LIN {X 0,Y 292.051,Z 857.28,A -85,B 0,C 180,E1 15092.157,E2 15092.157} C_VEL
LIN {X 0,Y 292.417,Z 857.28,A -85,B 0,C 180,E1 15098.753,E2 15098.753} C_VEL
LIN {X 0,Y 292.75,Z 857.28,A -85,B 0,C 180,E1 15104.981,E2 15104.981} C_VEL
LIN {X 0,Y 293.457,Z 857.28,A -85,B 0,C 180,E1 15114.042,E2 15114.042} C_VEL
LIN {X 0,Y 293.996,Z 857.28,A -85,B 0,C 180,E1 15119.962,E2 15119.962} C_VEL
LIN {X 0,Y 293.479,Z 857.28,A -85,B 0,C 180,E1 15125.882,E2 15125.882} C_VEL
LIN {X 0,Y 293.039,Z 857.28,A -85,B 0,C 180,E1 15131.883,E2 15131.883} C_VEL
LIN {X 0,Y 292.64,Z 857.28,A -85,B 0,C 180,E1 15138.037,E2 15138.037} C_VEL
LIN {X 0,Y 292.24,Z 857.28,A -85,B 0,C 180,E1 15144.433,E2 15144.433} C_VEL
LIN {X 0,Y 291.833,Z 857.307,A -85,B 0,C 180,E1 15152.49,E2 15152.49} C_VEL
LIN {X 0,Y 294.082,Z 862.737,A -85,B 0,C 180,E1 15153.268,E2 15153.268} C_VEL
LIN {X 0,Y 306.27,Z 885.121,A -85,B 0,C 180,E1 15157.392,E2 15157.392} C_VEL
LIN {X 0,Y 314.782,Z 908.516,A -85,B 0,C 180,E1 15161.429,E2 15161.429} C_VEL
LIN {X 0,Y 318.92,Z 932.003,A -85,B 0,C 180,E1 15165.576,E2 15165.576} C_VEL
LIN {X 0,Y 315.348,Z 948.213,A -85,B 0,C 180,E1 15168.226,E2 15168.226} C_VEL
LIN {X 0,Y 308.77,Z 968.688,A -85,B 0,C 180,E1 15172.765,E2 15172.765} C_VEL
LIN {X 0,Y 303.225,Z 983.739,A -85,B 0,C 180,E1 15177.978,E2 15177.978} C_VEL
LIN {X 0,Y 299.821,Z 992.395,A -85,B 0,C 180,E1 15182.966,E2 15182.966} C_VEL
LIN {X 0,Y 297.402,Z 997.125,A -85,B 0,C 180,E1 15189.121,E2 15189.121} C_VEL
LIN {X 0,Y 296.865,Z 995.934,A -85,B 0,C 180,E1 15195.459,E2 15195.459} C_VEL
LIN {X 0,Y 298.171,Z 989.36,A -85,B 0,C 180,E1 15201.237,E2 15201.237} C_VEL
LIN {X 0,Y 300.527,Z 978.42,A -85,B 0,C 180,E1 15206.388,E2 15206.388} C_VEL
LIN {X 0,Y 304.232,Z 961.601,A -85,B 0,C 180,E1 15211.425,E2 15211.425} C_VEL
LIN {X 0,Y 308.992,Z 939.449,A -85,B 0,C 180,E1 15215.799,E2 15215.799} C_VEL
LIN {X 0,Y 311.298,Z 922.827,A -85,B 0,C 180,E1 15218.213,E2 15218.213} C_VEL
LIN {X 0,Y 307.426,Z 899.704,A -85,B 0,C 180,E1 15221.361,E2 15221.361} C_VEL
LIN {X 0,Y 298.936,Z 872.735,A -85,B 0,C 180,E1 15224.452,E2 15224.452} C_VEL
LIN {X 0,Y 292.791,Z 857.28,A -85,B 0,C 180,E1 15226.014,E2 15226.014} C_VEL
LIN {X 0,Y 292.167,Z 857.28,A -85,B 0,C 180,E1 15234.492,E2 15234.492} C_VEL
LIN {X 0,Y 291.84,Z 857.28,A -85,B 0,C 180,E1 15241.251,E2 15241.251} C_VEL
LIN {X 0,Y 291.876,Z 857.28,A -85,B 0,C 180,E1 15249.731,E2 15249.731} C_VEL
LIN {X 0,Y 301.053,Z 889.147,A -85,B 0,C 180,E1 15251.908,E2 15251.908} C_VEL
LIN {X 0,Y 306.355,Z 915.006,A -85,B 0,C 180,E1 15254.516,E2 15254.516} C_VEL
LIN {X 0,Y 304.215,Z 939.148,A -85,B 0,C 180,E1 15257.526,E2 15257.526} C_VEL
LIN {X 0,Y 301.338,Z 961.008,A -85,B 0,C 180,E1 15261.49,E2 15261.49} C_VEL
LIN {X 0,Y 298.964,Z 978.431,A -85,B 0,C 180,E1 15266.207,E2 15266.207} C_VEL
LIN {X 0,Y 297.475,Z 990.318,A -85,B 0,C 180,E1 15271.29,E2 15271.29} C_VEL
LIN {X 0,Y 296.907,Z 996.961,A -85,B 0,C 180,E1 15276.62,E2 15276.62} C_VEL
LIN {X 0,Y 297.738,Z 998.146,A -85,B 0,C 180,E1 15282.282,E2 15282.282} C_VEL
LIN {X 0,Y 299.876,Z 993.695,A -85,B 0,C 180,E1 15287.652,E2 15287.652} C_VEL
LIN {X 0,Y 303.37,Z 983.119,A -85,B 0,C 180,E1 15293.016,E2 15293.016} C_VEL
LIN {X 0,Y 307.54,Z 967.861,A -85,B 0,C 180,E1 15297.568,E2 15297.568} C_VEL
LIN {X 0,Y 312.162,Z 947.905,A -85,B 0,C 180,E1 15301.439,E2 15301.439} C_VEL
LIN {X 0,Y 316.12,Z 922.658,A -85,B 0,C 180,E1 15304.704,E2 15304.704} C_VEL
LIN {X 0,Y 312.93,Z 899.843,A -85,B 0,C 180,E1 15307.526,E2 15307.526} C_VEL
LIN {X 0,Y 304.863,Z 879.144,A -85,B 0,C 180,E1 15310.308,E2 15310.308} C_VEL
LIN {X 0,Y 295.138,Z 862.737,A -85,B 0,C 180,E1 15313.251,E2 15313.251} C_VEL
LIN {X 0,Y 292.877,Z 857.28,A -85,B 0,C 180,E1 15314.248,E2 15314.248} C_VEL
LIN {X 0,Y 292.427,Z 857.28,A -85,B 0,C 180,E1 15321.281,E2 15321.281} C_VEL
LIN {X 0,Y 292.014,Z 857.28,A -85,B 0,C 180,E1 15328.186,E2 15328.186} C_VEL
LIN {X 0,Y 291.802,Z 857.28,A -85,B 0,C 180,E1 15334.832,E2 15334.832} C_VEL
LIN {X 0,Y 291.583,Z 857.28,A -85,B 0,C 180,E1 15343.369,E2 15343.369} C_VEL
LIN {X 0,Y 291.824,Z 857.28,A -85,B 0,C 180,E1 15347.489,E2 15347.489} C_VEL
LIN {X 0,Y 313.414,Z 909.451,A -85,B 0,C 180,E1 15351.464,E2 15351.464} C_VEL
LIN {X 0,Y 320.249,Z 933.058,A -85,B 0,C 180,E1 15353.265,E2 15353.265} C_VEL
LIN {X 0,Y 315.373,Z 966.492,A -85,B 0,C 180,E1 15355.452,E2 15355.452} C_VEL
LIN {X 0,Y 309.547,Z 998.009,A -85,B 0,C 180,E1 15358.778,E2 15358.778} C_VEL
LIN {X 0,Y 303.847,Z 1024.876,A -85,B 0,C 180,E1 15362.955,E2 15362.955} C_VEL
LIN {X 0,Y 299.229,Z 1047.786,A -85,B 0,C 180,E1 15368.09,E2 15368.09} C_VEL
LIN {X 0,Y 296.572,Z 1065.205,A -85,B 0,C 180,E1 15373.694,E2 15373.694} C_VEL
LIN {X 0,Y 295.641,Z 1077.565,A -85,B 0,C 180,E1 15379.675,E2 15379.675} C_VEL
LIN {X 0,Y 295.789,Z 1083.188,A -85,B 0,C 180,E1 15384.125,E2 15384.125} C_VEL
LIN {X 0,Y 296.066,Z 1086.174,A -85,B 0,C 180,E1 15390.001,E2 15390.001} C_VEL
LIN {X 0,Y 295.708,Z 1084.155,A -85,B 0,C 180,E1 15395.879,E2 15395.879} C_VEL
LIN {X 0,Y 295.5,Z 1077.25,A -85,B 0,C 180,E1 15401.828,E2 15401.828} C_VEL
LIN {X 0,Y 297.243,Z 1063.717,A -85,B 0,C 180,E1 15408.399,E2 15408.399} C_VEL
LIN {X 0,Y 301.566,Z 1044.337,A -85,B 0,C 180,E1 15414.543,E2 15414.543} C_VEL
LIN {X 0,Y 307.998,Z 1020.257,A -85,B 0,C 180,E1 15419.758,E2 15419.758} C_VEL
LIN {X 0,Y 315.4,Z 992.25,A -85,B 0,C 180,E1 15423.923,E2 15423.923} C_VEL
LIN {X 0,Y 322.553,Z 960.566,A -85,B 0,C 180,E1 15427.038,E2 15427.038} C_VEL
LIN {X 0,Y 326.962,Z 932.174,A -85,B 0,C 180,E1 15428.868,E2 15428.868} C_VEL
LIN {X 0,Y 318.461,Z 906.2,A -85,B 0,C 180,E1 15431.59,E2 15431.59} C_VEL
LIN {X 0,Y 317.145,Z 903.31,A -85,B 0,C 180,E1 15431.93,E2 15431.93} C_VEL
LIN {X 0,Y 310.668,Z 894.982,A -85,B 0,C 180,E1 15433.356,E2 15433.356} C_VEL
LIN {X 0,Y 299.831,Z 884.402,A -85,B 0,C 180,E1 15435.807,E2 15435.807} C_VEL
LIN {X 0,Y 298.921,Z 882.832,A -85,B 0,C 180,E1 15436.05,E2 15436.05} C_VEL
LIN {X 0,Y 286.284,Z 862.993,A -85,B 0,C 180,E1 15439.689,E2 15439.689} C_VEL
LIN {X 0,Y 283.795,Z 857.28,A -85,B 0,C 180,E1 15440.762,E2 15440.762} C_VEL
LIN {X 0,Y 283.97,Z 857.28,A -85,B 0,C 180,E1 15448.552,E2 15448.552} C_VEL
LIN {X 0,Y 284.238,Z 857.28,A -85,B 0,C 180,E1 15454.901,E2 15454.901} C_VEL
LIN {X 0,Y 284.673,Z 857.28,A -85,B 0,C 180,E1 15463.211,E2 15463.211} C_VEL
LIN {X 0,Y 285.234,Z 857.28,A -85,B 0,C 180,E1 15470.801,E2 15470.801} C_VEL
LIN {X 0,Y 285.877,Z 857.28,A -85,B 0,C 180,E1 15476.927,E2 15476.927} C_VEL
LIN {X 0,Y 285.868,Z 857.28,A -85,B 0,C 180,E1 15482.996,E2 15482.996} C_VEL
LIN {X 0,Y 285.075,Z 857.28,A -85,B 0,C 180,E1 15492.22,E2 15492.22} C_VEL
LIN {X 0,Y 284.66,Z 857.28,A -85,B 0,C 180,E1 15498.561,E2 15498.561} C_VEL
LIN {X 0,Y 284.213,Z 857.28,A -85,B 0,C 180,E1 15505.171,E2 15505.171} C_VEL
LIN {X 0,Y 283.965,Z 857.28,A -85,B 0,C 180,E1 15510.494,E2 15510.494} C_VEL
LIN {X 0,Y 286.238,Z 862.79,A -85,B 0,C 180,E1 15511.368,E2 15511.368} C_VEL
LIN {X 0,Y 298.239,Z 884.055,A -85,B 0,C 180,E1 15515.658,E2 15515.658} C_VEL
LIN {X 0,Y 307.422,Z 908.201,A -85,B 0,C 180,E1 15520.086,E2 15520.086} C_VEL
LIN {X 0,Y 311.823,Z 930.492,A -85,B 0,C 180,E1 15524.182,E2 15524.182} C_VEL
LIN {X 0,Y 311.465,Z 939.871,A -85,B 0,C 180,E1 15525.876,E2 15525.876} C_VEL
LIN {X 0,Y 304.54,Z 962.032,A -85,B 0,C 180,E1 15530.089,E2 15530.089} C_VEL
LIN {X 0,Y 298.43,Z 978.637,A -85,B 0,C 180,E1 15534.895,E2 15534.895} C_VEL
LIN {X 0,Y 293.676,Z 990.339,A -85,B 0,C 180,E1 15540.308,E2 15540.308} C_VEL
LIN {X 0,Y 290.878,Z 996.46,A -85,B 0,C 180,E1 15545.39,E2 15545.39} C_VEL
LIN {X 0,Y 289.12,Z 998.561,A -85,B 0,C 180,E1 15551.686,E2 15551.686} C_VEL
LIN {X 0,Y 289.394,Z 995.02,A -85,B 0,C 180,E1 15557.919,E2 15557.919} C_VEL
LIN {X 0,Y 291.487,Z 985.654,A -85,B 0,C 180,E1 15564.036,E2 15564.036} C_VEL
LIN {X 0,Y 294.927,Z 970.748,A -85,B 0,C 180,E1 15569.638,E2 15569.638} C_VEL
LIN {X 0,Y 299.377,Z 951.389,A -85,B 0,C 180,E1 15574.35,E2 15574.35} C_VEL
LIN {X 0,Y 304.25,Z 927.681,A -85,B 0,C 180,E1 15578.225,E2 15578.225} C_VEL
LIN {X 0,Y 300.861,Z 904.233,A -85,B 0,C 180,E1 15581.612,E2 15581.612} C_VEL
LIN {X 0,Y 292.909,Z 877.335,A -85,B 0,C 180,E1 15584.884,E2 15584.884} C_VEL
LIN {X 0,Y 284.754,Z 857.28,A -85,B 0,C 180,E1 15587.062,E2 15587.062} C_VEL
LIN {X 0,Y 284.152,Z 857.28,A -85,B 0,C 180,E1 15595.23,E2 15595.23} C_VEL
LIN {X 0,Y 283.876,Z 857.28,A -85,B 0,C 180,E1 15602.231,E2 15602.231} C_VEL
LIN {X 0,Y 283.938,Z 857.591,A -85,B 0,C 180,E1 15609.114,E2 15609.114} C_VEL
LIN {X 0,Y 292.917,Z 887.919,A -85,B 0,C 180,E1 15611.226,E2 15611.226} C_VEL
LIN {X 0,Y 298.57,Z 914.947,A -85,B 0,C 180,E1 15613.964,E2 15613.964} C_VEL
LIN {X 0,Y 297.666,Z 932.003,A -85,B 0,C 180,E1 15616.014,E2 15616.014} C_VEL
LIN {X 0,Y 294.567,Z 955.511,A -85,B 0,C 180,E1 15619.844,E2 15619.844} C_VEL
LIN {X 0,Y 291.757,Z 975.193,A -85,B 0,C 180,E1 15624.652,E2 15624.652} C_VEL
LIN {X 0,Y 290.044,Z 988.276,A -85,B 0,C 180,E1 15629.582,E2 15629.582} C_VEL
LIN {X 0,Y 289.1,Z 996.941,A -85,B 0,C 180,E1 15635.284,E2 15635.284} C_VEL
LIN {X 0,Y 289.475,Z 999.663,A -85,B 0,C 180,E1 15640.298,E2 15640.298} C_VEL
LIN {X 0,Y 291.556,Z 996.856,A -85,B 0,C 180,E1 15646.531,E2 15646.531} C_VEL
LIN {X 0,Y 294.757,Z 988.441,A -85,B 0,C 180,E1 15651.921,E2 15651.921} C_VEL
LIN {X 0,Y 299.092,Z 974.706,A -85,B 0,C 180,E1 15656.813,E2 15656.813} C_VEL
LIN {X 0,Y 304.047,Z 955.73,A -85,B 0,C 180,E1 15661.098,E2 15661.098} C_VEL
LIN {X 0,Y 308.919,Z 931.93,A -85,B 0,C 180,E1 15664.602,E2 15664.602} C_VEL
LIN {X 0,Y 309.271,Z 917.044,A -85,B 0,C 180,E1 15666.479,E2 15666.479} C_VEL
LIN {X 0,Y 304.585,Z 894.987,A -85,B 0,C 180,E1 15669.387,E2 15669.387} C_VEL
LIN {X 0,Y 294.414,Z 874.073,A -85,B 0,C 180,E1 15672.781,E2 15672.781} C_VEL
LIN {X 0,Y 287.331,Z 863.007,A -85,B 0,C 180,E1 15675.309,E2 15675.309} C_VEL
LIN {X 0,Y 284.773,Z 857.873,A -85,B 0,C 180,E1 15676.446,E2 15676.446} C_VEL
LIN {X 0,Y 284.247,Z 857.28,A -85,B 0,C 180,E1 15685.254,E2 15685.254} C_VEL
LIN {X 0,Y 283.918,Z 857.28,A -85,B 0,C 180,E1 15692.258,E2 15692.258} C_VEL
LIN {X 0,Y 283.636,Z 857.28,A -85,B 0,C 180,E1 15699.865,E2 15699.865} C_VEL
LIN {X 0,Y 283.896,Z 857.417,A -85,B 0,C 180,E1 15706.478,E2 15706.478} C_VEL
LIN {X 0,Y 305.889,Z 909.715,A -85,B 0,C 180,E1 15710.687,E2 15710.687} C_VEL
LIN {X 0,Y 313.023,Z 934.811,A -85,B 0,C 180,E1 15712.692,E2 15712.692} C_VEL
LIN {X 0,Y 308.007,Z 967.343,A -85,B 0,C 180,E1 15714.935,E2 15714.935} C_VEL
LIN {X 0,Y 302.051,Z 998.129,A -85,B 0,C 180,E1 15718.313,E2 15718.313} C_VEL
LIN {X 0,Y 296.162,Z 1024.75,A -85,B 0,C 180,E1 15722.607,E2 15722.607} C_VEL
LIN {X 0,Y 291.415,Z 1047.459,A -85,B 0,C 180,E1 15727.873,E2 15727.873} C_VEL
LIN {X 0,Y 288.578,Z 1065.563,A -85,B 0,C 180,E1 15734.012,E2 15734.012} C_VEL
LIN {X 0,Y 287.802,Z 1077.356,A -85,B 0,C 180,E1 15740.156,E2 15740.156} C_VEL
LIN {X 0,Y 287.912,Z 1083.164,A -85,B 0,C 180,E1 15745.477,E2 15745.477} C_VEL
LIN {X 0,Y 288.249,Z 1084.978,A -85,B 0,C 180,E1 15750.001,E2 15750.001} C_VEL
LIN {X 0,Y 287.855,Z 1083.014,A -85,B 0,C 180,E1 15756.04,E2 15756.04} C_VEL
LIN {X 0,Y 287.661,Z 1076.153,A -85,B 0,C 180,E1 15762.155,E2 15762.155} C_VEL
LIN {X 0,Y 289.488,Z 1063.13,A -85,B 0,C 180,E1 15768.729,E2 15768.729} C_VEL
LIN {X 0,Y 293.872,Z 1044.632,A -85,B 0,C 180,E1 15774.869,E2 15774.869} C_VEL
LIN {X 0,Y 300.588,Z 1020.977,A -85,B 0,C 180,E1 15780.247,E2 15780.247} C_VEL
LIN {X 0,Y 308.41,Z 992.884,A -85,B 0,C 180,E1 15784.587,E2 15784.587} C_VEL
LIN {X 0,Y 315.859,Z 961.774,A -85,B 0,C 180,E1 15787.763,E2 15787.763} C_VEL
LIN {X 0,Y 320.588,Z 934.743,A -85,B 0,C 180,E1 15789.585,E2 15789.585} C_VEL
LIN {X 0,Y 312.809,Z 909.957,A -85,B 0,C 180,E1 15792.355,E2 15792.355} C_VEL
LIN {X 0,Y 298.921,Z 882.832,A -85,B 0,C 180,E1 15796.05,E2 15796.05} C_VEL
LIN {X 0,Y 294.151,Z 878.708,A -85,B 0,C 180,E1 15797.228,E2 15797.228} C_VEL
LIN {X 0,Y 286.224,Z 874.597,A -85,B 0,C 180,E1 15799.245,E2 15799.245} C_VEL
LIN {X 0,Y 285.555,Z 873.708,A -85,B 0,C 180,E1 15799.446,E2 15799.446} C_VEL
LIN {X 0,Y 278.339,Z 862.989,A -85,B 0,C 180,E1 15801.827,E2 15801.827} C_VEL
LIN {X 0,Y 275.912,Z 858.523,A -85,B 0,C 180,E1 15802.729,E2 15802.729} C_VEL
LIN {X 0,Y 275.812,Z 857.28,A -85,B 0,C 180,E1 15802.822,E2 15802.822} C_VEL
LIN {X 0,Y 276.138,Z 857.28,A -85,B 0,C 180,E1 15811.319,E2 15811.319} C_VEL
LIN {X 0,Y 276.489,Z 857.28,A -85,B 0,C 180,E1 15818.584,E2 15818.584} C_VEL
LIN {X 0,Y 276.987,Z 857.28,A -85,B 0,C 180,E1 15827.335,E2 15827.335} C_VEL
LIN {X 0,Y 277.571,Z 857.28,A -85,B 0,C 180,E1 15833.699,E2 15833.699} C_VEL
LIN {X 0,Y 278.214,Z 857.28,A -85,B 0,C 180,E1 15839.96,E2 15839.96} C_VEL
LIN {X 0,Y 277.596,Z 857.28,A -85,B 0,C 180,E1 15846.22,E2 15846.22} C_VEL
LIN {X 0,Y 277.106,Z 857.28,A -85,B 0,C 180,E1 15852.578,E2 15852.578} C_VEL
LIN {X 0,Y 276.528,Z 857.28,A -85,B 0,C 180,E1 15861.436,E2 15861.436} C_VEL
LIN {X 0,Y 276.144,Z 857.447,A -85,B 0,C 180,E1 15868.317,E2 15868.317} C_VEL
LIN {X 0,Y 278.394,Z 862.813,A -85,B 0,C 180,E1 15869.246,E2 15869.246} C_VEL
LIN {X 0,Y 287.831,Z 878.44,A -85,B 0,C 180,E1 15872.812,E2 15872.812} C_VEL
LIN {X 0,Y 297.594,Z 899.927,A -85,B 0,C 180,E1 15877.132,E2 15877.132} C_VEL
LIN {X 0,Y 303.904,Z 923.425,A -85,B 0,C 180,E1 15881.64,E2 15881.64} C_VEL
LIN {X 0,Y 305.296,Z 940.028,A -85,B 0,C 180,E1 15884.9,E2 15884.9} C_VEL
LIN {X 0,Y 298.158,Z 962.047,A -85,B 0,C 180,E1 15889.086,E2 15889.086} C_VEL
LIN {X 0,Y 291.512,Z 979.299,A -85,B 0,C 180,E1 15894.083,E2 15894.083} C_VEL
LIN {X 0,Y 286.545,Z 990.786,A -85,B 0,C 180,E1 15899.357,E2 15899.357} C_VEL
LIN {X 0,Y 283.159,Z 997.767,A -85,B 0,C 180,E1 15905.22,E2 15905.22} C_VEL
LIN {X 0,Y 281.371,Z 999.797,A -85,B 0,C 180,E1 15911.163,E2 15911.163} C_VEL
LIN {X 0,Y 281.504,Z 996.586,A -85,B 0,C 180,E1 15917.575,E2 15917.575} C_VEL
LIN {X 0,Y 283.583,Z 987.566,A -85,B 0,C 180,E1 15923.869,E2 15923.869} C_VEL
LIN {X 0,Y 287.003,Z 973.119,A -85,B 0,C 180,E1 15929.621,E2 15929.621} C_VEL
LIN {X 0,Y 291.516,Z 954.311,A -85,B 0,C 180,E1 15934.467,E2 15934.467} C_VEL
LIN {X 0,Y 296.78,Z 930.157,A -85,B 0,C 180,E1 15938.618,E2 15938.618} C_VEL
LIN {X 0,Y 294.256,Z 908.622,A -85,B 0,C 180,E1 15941.876,E2 15941.876} C_VEL
LIN {X 0,Y 286.962,Z 882.251,A -85,B 0,C 180,E1 15945.295,E2 15945.295} C_VEL
LIN {X 0,Y 276.717,Z 857.28,A -85,B 0,C 180,E1 15948.168,E2 15948.168} C_VEL
LIN {X 0,Y 276.119,Z 857.28,A -85,B 0,C 180,E1 15956.018,E2 15956.018} C_VEL
LIN {X 0,Y 275.743,Z 857.28,A -85,B 0,C 180,E1 15964.657,E2 15964.657} C_VEL
LIN {X 0,Y 275.968,Z 857.28,A -85,B 0,C 180,E1 15968.419,E2 15968.419} C_VEL
LIN {X 0,Y 285.494,Z 889.664,A -85,B 0,C 180,E1 15970.765,E2 15970.765} C_VEL
LIN {X 0,Y 291.2,Z 917.429,A -85,B 0,C 180,E1 15973.701,E2 15973.701} C_VEL
LIN {X 0,Y 288.925,Z 941.854,A -85,B 0,C 180,E1 15976.917,E2 15976.917} C_VEL
LIN {X 0,Y 285.705,Z 964.372,A -85,B 0,C 180,E1 15981.246,E2 15981.246} C_VEL
LIN {X 0,Y 283.381,Z 980.958,A -85,B 0,C 180,E1 15986.028,E2 15986.028} C_VEL
LIN {X 0,Y 281.845,Z 992.463,A -85,B 0,C 180,E1 15991.146,E2 15991.146} C_VEL
LIN {X 0,Y 281.271,Z 998.914,A -85,B 0,C 180,E1 15996.218,E2 15996.218} C_VEL
LIN {X 0,Y 281.876,Z 1001.013,A -85,B 0,C 180,E1 16001.249,E2 16001.249} C_VEL
LIN {X 0,Y 283.6,Z 998.938,A -85,B 0,C 180,E1 16006.145,E2 16006.145} C_VEL
LIN {X 0,Y 286.889,Z 991.422,A -85,B 0,C 180,E1 16011.698,E2 16011.698} C_VEL
LIN {X 0,Y 291.641,Z 977.605,A -85,B 0,C 180,E1 16017.063,E2 16017.063} C_VEL
LIN {X 0,Y 297.012,Z 958.793,A -85,B 0,C 180,E1 16021.567,E2 16021.567} C_VEL
LIN {X 0,Y 302.322,Z 935.135,A -85,B 0,C 180,E1 16025.243,E2 16025.243} C_VEL
LIN {X 0,Y 303.209,Z 921.956,A -85,B 0,C 180,E1 16026.947,E2 16026.947} C_VEL
LIN {X 0,Y 299.526,Z 900.362,A -85,B 0,C 180,E1 16029.954,E2 16029.954} C_VEL
LIN {X 0,Y 290.435,Z 880.101,A -85,B 0,C 180,E1 16033.405,E2 16033.405} C_VEL
LIN {X 0,Y 283.088,Z 868.605,A -85,B 0,C 180,E1 16036.212,E2 16036.212} C_VEL
LIN {X 0,Y 279.789,Z 863.502,A -85,B 0,C 180,E1 16037.708,E2 16037.708} C_VEL
LIN {X 0,Y 276.691,Z 858.449,A -85,B 0,C 180,E1 16039.338,E2 16039.338} C_VEL
LIN {X 0,Y 276.551,Z 857.28,A -85,B 0,C 180,E1 16039.762,E2 16039.762} C_VEL
LIN {X 0,Y 276.14,Z 857.28,A -85,B 0,C 180,E1 16048.686,E2 16048.686} C_VEL
LIN {X 0,Y 275.737,Z 857.28,A -85,B 0,C 180,E1 16057.189,E2 16057.189} C_VEL
LIN {X 0,Y 275.834,Z 857.28,A -85,B 0,C 180,E1 16065.329,E2 16065.329} C_VEL
LIN {X 0,Y 297.764,Z 908.33,A -85,B 0,C 180,E1 16069.733,E2 16069.733} C_VEL
LIN {X 0,Y 305.82,Z 936.459,A -85,B 0,C 180,E1 16072.115,E2 16072.115} C_VEL
LIN {X 0,Y 300.666,Z 968.088,A -85,B 0,C 180,E1 16074.392,E2 16074.392} C_VEL
LIN {X 0,Y 294.64,Z 997.906,A -85,B 0,C 180,E1 16077.782,E2 16077.782} C_VEL
LIN {X 0,Y 288.312,Z 1025.453,A -85,B 0,C 180,E1 16082.41,E2 16082.41} C_VEL
LIN {X 0,Y 283.332,Z 1048.374,A -85,B 0,C 180,E1 16088.034,E2 16088.034} C_VEL
LIN {X 0,Y 280.588,Z 1065.886,A -85,B 0,C 180,E1 16094.348,E2 16094.348} C_VEL
LIN {X 0,Y 279.997,Z 1077.064,A -85,B 0,C 180,E1 16100.665,E2 16100.665} C_VEL
LIN {X 0,Y 280.196,Z 1082.833,A -85,B 0,C 180,E1 16106.904,E2 16106.904} C_VEL
LIN {X 0,Y 280.445,Z 1083.787,A -85,B 0,C 180,E1 16110.001,E2 16110.001} C_VEL
LIN {X 0,Y 280.005,Z 1081.875,A -85,B 0,C 180,E1 16116.21,E2 16116.21} C_VEL
LIN {X 0,Y 279.926,Z 1074.108,A -85,B 0,C 180,E1 16123.129,E2 16123.129} C_VEL
LIN {X 0,Y 282.241,Z 1060.018,A -85,B 0,C 180,E1 16130.135,E2 16130.135} C_VEL
LIN {X 0,Y 287.413,Z 1040.691,A -85,B 0,C 180,E1 16136.384,E2 16136.384} C_VEL
LIN {X 0,Y 294.216,Z 1018.216,A -85,B 0,C 180,E1 16141.4,E2 16141.4} C_VEL
LIN {X 0,Y 302.188,Z 990.915,A -85,B 0,C 180,E1 16145.625,E2 16145.625} C_VEL
LIN {X 0,Y 309.866,Z 960.253,A -85,B 0,C 180,E1 16148.749,E2 16148.749} C_VEL
LIN {X 0,Y 314.144,Z 936.628,A -85,B 0,C 180,E1 16150.391,E2 16150.391} C_VEL
LIN {X 0,Y 306.056,Z 910.819,A -85,B 0,C 180,E1 16153.501,E2 16153.501} C_VEL
LIN {X 0,Y 292.111,Z 884.189,A -85,B 0,C 180,E1 16157.483,E2 16157.483} C_VEL
LIN {X 0,Y 285.555,Z 873.708,A -85,B 0,C 180,E1 16159.446,E2 16159.446} C_VEL
LIN {X 0,Y 280.767,Z 870.562,A -85,B 0,C 180,E1 16160.828,E2 16160.828} C_VEL
LIN {X 0,Y 273.463,Z 867.295,A -85,B 0,C 180,E1 16163.063,E2 16163.063} C_VEL
LIN {X 0,Y 272.905,Z 866.38,A -85,B 0,C 180,E1 16163.275,E2 16163.275} C_VEL
LIN {X 0,Y 268.051,Z 858.961,A -85,B 0,C 180,E1 16165.179,E2 16165.179} C_VEL
LIN {X 0,Y 267.888,Z 857.28,A -85,B 0,C 180,E1 16165.551,E2 16165.551} C_VEL
LIN {X 0,Y 268.274,Z 857.28,A -85,B 0,C 180,E1 16174.558,E2 16174.558} C_VEL
LIN {X 0,Y 268.784,Z 857.28,A -85,B 0,C 180,E1 16183.264,E2 16183.264} C_VEL
LIN {X 0,Y 269.335,Z 857.28,A -85,B 0,C 180,E1 16190.253,E2 16190.253} C_VEL
LIN {X 0,Y 270.023,Z 857.28,A -85,B 0,C 180,E1 16196.746,E2 16196.746} C_VEL
LIN {X 0,Y 270.018,Z 857.28,A -85,B 0,C 180,E1 16203.172,E2 16203.172} C_VEL
LIN {X 0,Y 269.394,Z 857.28,A -85,B 0,C 180,E1 16209.661,E2 16209.661} C_VEL
LIN {X 0,Y 268.86,Z 857.28,A -85,B 0,C 180,E1 16216.79,E2 16216.79} C_VEL
LIN {X 0,Y 268.318,Z 857.8,A -85,B 0,C 180,E1 16225.871,E2 16225.871} C_VEL
LIN {X 0,Y 270.698,Z 863.025,A -85,B 0,C 180,E1 16226.936,E2 16226.936} C_VEL
LIN {X 0,Y 273.168,Z 866.494,A -85,B 0,C 180,E1 16227.907,E2 16227.907} C_VEL
LIN {X 0,Y 284.799,Z 886.727,A -85,B 0,C 180,E1 16232.796,E2 16232.796} C_VEL
LIN {X 0,Y 293.806,Z 910.224,A -85,B 0,C 180,E1 16237.664,E2 16237.664} C_VEL
LIN {X 0,Y 298.09,Z 931.36,A -85,B 0,C 180,E1 16241.943,E2 16241.943} C_VEL
LIN {X 0,Y 298.354,Z 943.061,A -85,B 0,C 180,E1 16244.335,E2 16244.335} C_VEL
LIN {X 0,Y 290.769,Z 964.901,A -85,B 0,C 180,E1 16248.702,E2 16248.702} C_VEL
LIN {X 0,Y 283.639,Z 982.168,A -85,B 0,C 180,E1 16254.041,E2 16254.041} C_VEL
LIN {X 0,Y 278.444,Z 993.5,A -85,B 0,C 180,E1 16259.803,E2 16259.803} C_VEL
LIN {X 0,Y 275.014,Z 999.728,A -85,B 0,C 180,E1 16266.026,E2 16266.026} C_VEL
LIN {X 0,Y 273.652,Z 1000.974,A -85,B 0,C 180,E1 16270.61,E2 16270.61} C_VEL
LIN {X 0,Y 273.613,Z 998.078,A -85,B 0,C 180,E1 16277.211,E2 16277.211} C_VEL
LIN {X 0,Y 275.688,Z 989.447,A -85,B 0,C 180,E1 16283.693,E2 16283.693} C_VEL
LIN {X 0,Y 279.054,Z 975.469,A -85,B 0,C 180,E1 16289.61,E2 16289.61} C_VEL
LIN {X 0,Y 283.673,Z 957.21,A -85,B 0,C 180,E1 16294.591,E2 16294.591} C_VEL
LIN {X 0,Y 289.064,Z 933.857,A -85,B 0,C 180,E1 16298.85,E2 16298.85} C_VEL
LIN {X 0,Y 288.727,Z 919.658,A -85,B 0,C 180,E1 16301.095,E2 16301.095} C_VEL
LIN {X 0,Y 283.06,Z 894.067,A -85,B 0,C 180,E1 16304.788,E2 16304.788} C_VEL
LIN {X 0,Y 273.024,Z 867.509,A -85,B 0,C 180,E1 16308.16,E2 16308.16} C_VEL
LIN {X 0,Y 268.655,Z 857.28,A -85,B 0,C 180,E1 16309.466,E2 16309.466} C_VEL
LIN {X 0,Y 268.145,Z 857.28,A -85,B 0,C 180,E1 16316.853,E2 16316.853} C_VEL
LIN {X 0,Y 267.818,Z 857.28,A -85,B 0,C 180,E1 16325.837,E2 16325.837} C_VEL
LIN {X 0,Y 268.002,Z 857.687,A -85,B 0,C 180,E1 16327.79,E2 16327.79} C_VEL
LIN {X 0,Y 277.552,Z 889.396,A -85,B 0,C 180,E1 16330.118,E2 16330.118} C_VEL
LIN {X 0,Y 283.33,Z 916.645,A -85,B 0,C 180,E1 16333.019,E2 16333.019} C_VEL
LIN {X 0,Y 283.104,Z 929.719,A -85,B 0,C 180,E1 16334.637,E2 16334.637} C_VEL
LIN {X 0,Y 279.619,Z 954.797,A -85,B 0,C 180,E1 16338.666,E2 16338.666} C_VEL
LIN {X 0,Y 276.664,Z 974.466,A -85,B 0,C 180,E1 16343.398,E2 16343.398} C_VEL
LIN {X 0,Y 274.61,Z 988.895,A -85,B 0,C 180,E1 16348.678,E2 16348.678} C_VEL
LIN {X 0,Y 273.587,Z 997.489,A -85,B 0,C 180,E1 16353.779,E2 16353.779} C_VEL
LIN {X 0,Y 273.829,Z 1002.126,A -85,B 0,C 180,E1 16360.045,E2 16360.045} C_VEL
LIN {X 0,Y 275.705,Z 1000.856,A -85,B 0,C 180,E1 16365.829,E2 16365.829} C_VEL
LIN {X 0,Y 278.943,Z 994.26,A -85,B 0,C 180,E1 16371.459,E2 16371.459} C_VEL
LIN {X 0,Y 283.889,Z 981.537,A -85,B 0,C 180,E1 16376.983,E2 16376.983} C_VEL
LIN {X 0,Y 289.496,Z 963.933,A -85,B 0,C 180,E1 16381.631,E2 16381.631} C_VEL
LIN {X 0,Y 295.178,Z 941.093,A -85,B 0,C 180,E1 16385.554,E2 16385.554} C_VEL
LIN {X 0,Y 297.132,Z 926.214,A -85,B 0,C 180,E1 16387.537,E2 16387.537} C_VEL
LIN {X 0,Y 294.198,Z 904.905,A -85,B 0,C 180,E1 16390.66,E2 16390.66} C_VEL
LIN {X 0,Y 286.161,Z 885.588,A -85,B 0,C 180,E1 16394.172,E2 16394.172} C_VEL
LIN {X 0,Y 277.161,Z 870.723,A -85,B 0,C 180,E1 16398.081,E2 16398.081} C_VEL
LIN {X 0,Y 272.471,Z 864.062,A -85,B 0,C 180,E1 16400.682,E2 16400.682} C_VEL
LIN {X 0,Y 268.495,Z 858.568,A -85,B 0,C 180,E1 16403.551,E2 16403.551} C_VEL
LIN {X 0,Y 268.292,Z 857.28,A -85,B 0,C 180,E1 16404.375,E2 16404.375} C_VEL
LIN {X 0,Y 267.903,Z 857.28,A -85,B 0,C 180,E1 16412.036,E2 16412.036} C_VEL
LIN {X 0,Y 267.816,Z 857.536,A -85,B 0,C 180,E1 16421.008,E2 16421.008} C_VEL
LIN {X 0,Y 269.952,Z 862.741,A -85,B 0,C 180,E1 16423.055,E2 16423.055} C_VEL
LIN {X 0,Y 272.275,Z 864.914,A -85,B 0,C 180,E1 16424.518,E2 16424.518} C_VEL
LIN {X 0,Y 274.414,Z 871.592,A -85,B 0,C 180,E1 16425.582,E2 16425.582} C_VEL
LIN {X 0,Y 291.505,Z 912.197,A -85,B 0,C 180,E1 16429.175,E2 16429.175} C_VEL
LIN {X 0,Y 298.596,Z 938.322,A -85,B 0,C 180,E1 16431.523,E2 16431.523} C_VEL
LIN {X 0,Y 293.02,Z 970.545,A -85,B 0,C 180,E1 16434.003,E2 16434.003} C_VEL
LIN {X 0,Y 286.791,Z 999.866,A -85,B 0,C 180,E1 16437.538,E2 16437.538} C_VEL
LIN {X 0,Y 280.285,Z 1026.873,A -85,B 0,C 180,E1 16442.36,E2 16442.36} C_VEL
LIN {X 0,Y 275.38,Z 1048.716,A -85,B 0,C 180,E1 16448.04,E2 16448.04} C_VEL
LIN {X 0,Y 272.671,Z 1065.611,A -85,B 0,C 180,E1 16454.487,E2 16454.487} C_VEL
LIN {X 0,Y 272.133,Z 1075.694,A -85,B 0,C 180,E1 16460.393,E2 16460.393} C_VEL
LIN {X 0,Y 272.378,Z 1081.583,A -85,B 0,C 180,E1 16466.815,E2 16466.815} C_VEL
LIN {X 0,Y 272.61,Z 1082.601,A -85,B 0,C 180,E1 16470.162,E2 16470.162} C_VEL
LIN {X 0,Y 272.126,Z 1080.735,A -85,B 0,C 180,E1 16476.39,E2 16476.39} C_VEL
LIN {X 0,Y 272.075,Z 1073.038,A -85,B 0,C 180,E1 16483.515,E2 16483.515} C_VEL
LIN {X 0,Y 274.525,Z 1059.393,A -85,B 0,C 180,E1 16490.562,E2 16490.562} C_VEL
LIN {X 0,Y 280.14,Z 1039.788,A -85,B 0,C 180,E1 16497.124,E2 16497.124} C_VEL
LIN {X 0,Y 287.797,Z 1015.949,A -85,B 0,C 180,E1 16502.524,E2 16502.524} C_VEL
LIN {X 0,Y 296.101,Z 988.908,A -85,B 0,C 180,E1 16506.701,E2 16506.701} C_VEL
LIN {X 0,Y 304.169,Z 957.852,A -85,B 0,C 180,E1 16509.852,E2 16509.852} C_VEL
LIN {X 0,Y 307.875,Z 939.161,A -85,B 0,C 180,E1 16511.166,E2 16511.166} C_VEL
LIN {X 0,Y 300.32,Z 914.342,A -85,B 0,C 180,E1 16514.357,E2 16514.357} C_VEL
LIN {X 0,Y 287.637,Z 889.171,A -85,B 0,C 180,E1 16518.335,E2 16518.335} C_VEL
LIN {X 0,Y 274.951,Z 869.364,A -85,B 0,C 180,E1 16522.526,E2 16522.526} C_VEL
LIN {X 0,Y 272.905,Z 866.38,A -85,B 0,C 180,E1 16523.275,E2 16523.275} C_VEL
LIN {X 0,Y 268.591,Z 863.637,A -85,B 0,C 180,E1 16524.773,E2 16524.773} C_VEL
LIN {X 0,Y 261.658,Z 862.121,A -85,B 0,C 180,E1 16527.298,E2 16527.298} C_VEL
LIN {X 0,Y 261.102,Z 861.355,A -85,B 0,C 180,E1 16527.553,E2 16527.553} C_VEL
LIN {X 0,Y 260.015,Z 857.28,A -85,B 0,C 180,E1 16528.359,E2 16528.359} C_VEL
LIN {X 0,Y 260.405,Z 857.28,A -85,B 0,C 180,E1 16535.948,E2 16535.948} C_VEL
LIN {X 0,Y 260.864,Z 857.28,A -85,B 0,C 180,E1 16543.093,E2 16543.093} C_VEL
LIN {X 0,Y 261.379,Z 857.28,A -85,B 0,C 180,E1 16549.987,E2 16549.987} C_VEL
LIN {X 0,Y 262.089,Z 857.28,A -85,B 0,C 180,E1 16556.647,E2 16556.647} C_VEL
LIN {X 0,Y 262.086,Z 857.28,A -85,B 0,C 180,E1 16563.268,E2 16563.268} C_VEL
LIN {X 0,Y 261.412,Z 857.28,A -85,B 0,C 180,E1 16570.052,E2 16570.052} C_VEL
LIN {X 0,Y 260.955,Z 857.28,A -85,B 0,C 180,E1 16576.812,E2 16576.812} C_VEL
LIN {X 0,Y 260.506,Z 857.479,A -85,B 0,C 180,E1 16582.991,E2 16582.991} C_VEL
LIN {X 0,Y 262.596,Z 862.754,A -85,B 0,C 180,E1 16584.101,E2 16584.101} C_VEL
LIN {X 0,Y 265.335,Z 866.104,A -85,B 0,C 180,E1 16585.318,E2 16585.318} C_VEL
LIN {X 0,Y 276.063,Z 884.195,A -85,B 0,C 180,E1 16590.197,E2 16590.197} C_VEL
LIN {X 0,Y 285.344,Z 905.868,A -85,B 0,C 180,E1 16595.178,E2 16595.178} C_VEL
LIN {X 0,Y 290.817,Z 927.564,A -85,B 0,C 180,E1 16599.809,E2 16599.809} C_VEL
LIN {X 0,Y 291.958,Z 944.294,A -85,B 0,C 180,E1 16603.444,E2 16603.444} C_VEL
LIN {X 0,Y 284.14,Z 965.961,A -85,B 0,C 180,E1 16607.868,E2 16607.868} C_VEL
LIN {X 0,Y 276.945,Z 982.514,A -85,B 0,C 180,E1 16613.03,E2 16613.03} C_VEL
LIN {X 0,Y 271.252,Z 994.156,A -85,B 0,C 180,E1 16618.913,E2 16618.913} C_VEL
LIN {X 0,Y 267.773,Z 1000.261,A -85,B 0,C 180,E1 16624.632,E2 16624.632} C_VEL
LIN {X 0,Y 265.966,Z 1002.151,A -85,B 0,C 180,E1 16630.027,E2 16630.027} C_VEL
LIN {X 0,Y 265.73,Z 999.558,A -85,B 0,C 180,E1 16636.825,E2 16636.825} C_VEL
LIN {X 0,Y 267.779,Z 991.249,A -85,B 0,C 180,E1 16643.506,E2 16643.506} C_VEL
LIN {X 0,Y 271.13,Z 977.705,A -85,B 0,C 180,E1 16649.599,E2 16649.599} C_VEL
LIN {X 0,Y 275.791,Z 959.971,A -85,B 0,C 180,E1 16654.723,E2 16654.723} C_VEL
LIN {X 0,Y 281.636,Z 936.25,A -85,B 0,C 180,E1 16659.28,E2 16659.28} C_VEL
LIN {X 0,Y 281.901,Z 924.382,A -85,B 0,C 180,E1 16661.226,E2 16661.226} C_VEL
LIN {X 0,Y 277.153,Z 899.865,A -85,B 0,C 180,E1 16664.984,E2 16664.984} C_VEL
LIN {X 0,Y 268.187,Z 874.473,A -85,B 0,C 180,E1 16668.452,E2 16668.452} C_VEL
LIN {X 0,Y 260.54,Z 857.28,A -85,B 0,C 180,E1 16670.729,E2 16670.729} C_VEL
LIN {X 0,Y 259.998,Z 857.28,A -85,B 0,C 180,E1 16679.263,E2 16679.263} C_VEL
LIN {X 0,Y 259.994,Z 857.28,A -85,B 0,C 180,E1 16687.002,E2 16687.002} C_VEL
LIN {X 0,Y 270.165,Z 891.19,A -85,B 0,C 180,E1 16689.636,E2 16689.636} C_VEL
LIN {X 0,Y 275.933,Z 919.004,A -85,B 0,C 180,E1 16692.725,E2 16692.725} C_VEL
LIN {X 0,Y 274.579,Z 937.182,A -85,B 0,C 180,E1 16695.111,E2 16695.111} C_VEL
LIN {X 0,Y 271.357,Z 959.8,A -85,B 0,C 180,E1 16699.176,E2 16699.176} C_VEL
LIN {X 0,Y 268.328,Z 979.229,A -85,B 0,C 180,E1 16704.359,E2 16704.359} C_VEL
LIN {X 0,Y 266.336,Z 993.415,A -85,B 0,C 180,E1 16710.337,E2 16710.337} C_VEL
LIN {X 0,Y 265.624,Z 1001.408,A -85,B 0,C 180,E1 16716.54,E2 16716.54} C_VEL
LIN {X 0,Y 266.029,Z 1003.337,A -85,B 0,C 180,E1 16720.086,E2 16720.086} C_VEL
LIN {X 0,Y 267.283,Z 1003.169,A -85,B 0,C 180,E1 16724.361,E2 16724.361} C_VEL
LIN {X 0,Y 270.456,Z 998.194,A -85,B 0,C 180,E1 16730.377,E2 16730.377} C_VEL
LIN {X 0,Y 275.455,Z 986.874,A -85,B 0,C 180,E1 16736.309,E2 16736.309} C_VEL
LIN {X 0,Y 281.109,Z 971.293,A -85,B 0,C 180,E1 16741.13,E2 16741.13} C_VEL
LIN {X 0,Y 287.211,Z 950.312,A -85,B 0,C 180,E1 16745.33,E2 16745.33} C_VEL
LIN {X 0,Y 291.102,Z 929.739,A -85,B 0,C 180,E1 16748.253,E2 16748.253} C_VEL
LIN {X 0,Y 289.06,Z 909.862,A -85,B 0,C 180,E1 16751.328,E2 16751.328} C_VEL
LIN {X 0,Y 282.05,Z 891.22,A -85,B 0,C 180,E1 16754.929,E2 16754.929} C_VEL
LIN {X 0,Y 273.87,Z 877.295,A -85,B 0,C 180,E1 16758.8,E2 16758.8} C_VEL
LIN {X 0,Y 269.495,Z 870.966,A -85,B 0,C 180,E1 16761.41,E2 16761.41} C_VEL
LIN {X 0,Y 265.427,Z 864.63,A -85,B 0,C 180,E1 16764.834,E2 16764.834} C_VEL
LIN {X 0,Y 261.36,Z 861.647,A -85,B 0,C 180,E1 16771.459,E2 16771.459} C_VEL
LIN {X 0,Y 263.508,Z 863.923,A -85,B 0,C 180,E1 16778.4,E2 16778.4} C_VEL
LIN {X 0,Y 265.602,Z 865.687,A -85,B 0,C 180,E1 16780.599,E2 16780.599} C_VEL
LIN {X 0,Y 269.602,Z 872.807,A -85,B 0,C 180,E1 16784.003,E2 16784.003} C_VEL
LIN {X 0,Y 271.519,Z 882.157,A -85,B 0,C 180,E1 16785.49,E2 16785.49} C_VEL
LIN {X 0,Y 285.608,Z 917.378,A -85,B 0,C 180,E1 16788.736,E2 16788.736} C_VEL
LIN {X 0,Y 291.331,Z 940.698,A -85,B 0,C 180,E1 16790.941,E2 16790.941} C_VEL
LIN {X 0,Y 285.232,Z 973.572,A -85,B 0,C 180,E1 16793.663,E2 16793.663} C_VEL
LIN {X 0,Y 278.5,Z 1003.205,A -85,B 0,C 180,E1 16797.531,E2 16797.531} C_VEL
LIN {X 0,Y 272.268,Z 1028.093,A -85,B 0,C 180,E1 16802.29,E2 16802.29} C_VEL
LIN {X 0,Y 267.482,Z 1048.685,A -85,B 0,C 180,E1 16807.937,E2 16807.937} C_VEL
LIN {X 0,Y 264.881,Z 1064.564,A -85,B 0,C 180,E1 16814.247,E2 16814.247} C_VEL
LIN {X 0,Y 264.301,Z 1075.379,A -85,B 0,C 180,E1 16820.937,E2 16820.937} C_VEL
LIN {X 0,Y 264.554,Z 1080.328,A -85,B 0,C 180,E1 16826.72,E2 16826.72} C_VEL
LIN {X 0,Y 264.819,Z 1081.398,A -85,B 0,C 180,E1 16830.001,E2 16830.001} C_VEL
LIN {X 0,Y 264.275,Z 1079.601,A -85,B 0,C 180,E1 16836.581,E2 16836.581} C_VEL
LIN {X 0,Y 264.163,Z 1072.9,A -85,B 0,C 180,E1 16843.255,E2 16843.255} C_VEL
LIN {X 0,Y 266.291,Z 1061.171,A -85,B 0,C 180,E1 16849.948,E2 16849.948} C_VEL
LIN {X 0,Y 271.407,Z 1043.656,A -85,B 0,C 180,E1 16856.507,E2 16856.507} C_VEL
LIN {X 0,Y 279.283,Z 1020.421,A -85,B 0,C 180,E1 16862.369,E2 16862.369} C_VEL
LIN {X 0,Y 288.125,Z 993.526,A -85,B 0,C 180,E1 16866.945,E2 16866.945} C_VEL
LIN {X 0,Y 296.743,Z 963.024,A -85,B 0,C 180,E1 16870.362,E2 16870.362} C_VEL
LIN {X 0,Y 301.485,Z 941.062,A -85,B 0,C 180,E1 16872.034,E2 16872.034} C_VEL
LIN {X 0,Y 293.993,Z 916.028,A -85,B 0,C 180,E1 16875.492,E2 16875.492} C_VEL
LIN {X 0,Y 281.483,Z 891.242,A -85,B 0,C 180,E1 16879.768,E2 16879.768} C_VEL
LIN {X 0,Y 268.225,Z 870.575,A -85,B 0,C 180,E1 16884.553,E2 16884.553} C_VEL
LIN {X 0,Y 263.055,Z 863.569,A -85,B 0,C 180,E1 16886.693,E2 16886.693} C_VEL
LIN {X 0,Y 261.102,Z 861.355,A -85,B 0,C 180,E1 16887.553,E2 16887.553} C_VEL
LIN {X 0,Y 256.137,Z 857.592,A -85,B 0,C 180,E1 16889.802,E2 16889.802} C_VEL
LIN {X 0,Y 252.223,Z 857.28,A -85,B 0,C 180,E1 16892.374,E2 16892.374} C_VEL
LIN {X 0,Y 252.631,Z 857.28,A -85,B 0,C 180,E1 16898.887,E2 16898.887} C_VEL
LIN {X 0,Y 253.084,Z 857.28,A -85,B 0,C 180,E1 16906.116,E2 16906.116} C_VEL
LIN {X 0,Y 253.771,Z 857.28,A -85,B 0,C 180,E1 16913.106,E2 16913.106} C_VEL
LIN {X 0,Y 254.513,Z 857.28,A -85,B 0,C 180,E1 16919.956,E2 16919.956} C_VEL
LIN {X 0,Y 253.798,Z 857.28,A -85,B 0,C 180,E1 16926.805,E2 16926.805} C_VEL
LIN {X 0,Y 253.2,Z 857.28,A -85,B 0,C 180,E1 16933.788,E2 16933.788} C_VEL
LIN {X 0,Y 252.742,Z 857.28,A -85,B 0,C 180,E1 16939.637,E2 16939.637} C_VEL
LIN {X 0,Y 254.759,Z 862.642,A -85,B 0,C 180,E1 16940.912,E2 16940.912} C_VEL
LIN {X 0,Y 257.728,Z 865.989,A -85,B 0,C 180,E1 16942.411,E2 16942.411} C_VEL
LIN {X 0,Y 268.602,Z 883.643,A -85,B 0,C 180,E1 16947.881,E2 16947.881} C_VEL
LIN {X 0,Y 278.438,Z 906.126,A -85,B 0,C 180,E1 16953.506,E2 16953.506} C_VEL
LIN {X 0,Y 283.932,Z 927.419,A -85,B 0,C 180,E1 16958.323,E2 16958.323} C_VEL
LIN {X 0,Y 285.306,Z 946.874,A -85,B 0,C 180,E1 16962.747,E2 16962.747} C_VEL
LIN {X 0,Y 276.746,Z 968.865,A -85,B 0,C 180,E1 16967.469,E2 16967.469} C_VEL
LIN {X 0,Y 269.291,Z 984.962,A -85,B 0,C 180,E1 16972.812,E2 16972.812} C_VEL
LIN {X 0,Y 263.483,Z 996.099,A -85,B 0,C 180,E1 16978.856,E2 16978.856} C_VEL
LIN {X 0,Y 259.444,Z 1002.392,A -85,B 0,C 180,E1 16985.887,E2 16985.887} C_VEL
LIN {X 0,Y 257.779,Z 1002.876,A -85,B 0,C 180,E1 16992.92,E2 16992.92} C_VEL
LIN {X 0,Y 258.575,Z 997.788,A -85,B 0,C 180,E1 16999.881,E2 16999.881} C_VEL
LIN {X 0,Y 261.488,Z 986.793,A -85,B 0,C 180,E1 17006.679,E2 17006.679} C_VEL
LIN {X 0,Y 265.994,Z 970.262,A -85,B 0,C 180,E1 17012.792,E2 17012.792} C_VEL
LIN {X 0,Y 271.256,Z 950.349,A -85,B 0,C 180,E1 17017.617,E2 17017.617} C_VEL
LIN {X 0,Y 275.159,Z 931.818,A -85,B 0,C 180,E1 17020.844,E2 17020.844} C_VEL
LIN {X 0,Y 271.731,Z 908.507,A -85,B 0,C 180,E1 17024.725,E2 17024.725} C_VEL
LIN {X 0,Y 264.106,Z 883.368,A -85,B 0,C 180,E1 17028.419,E2 17028.419} C_VEL
LIN {X 0,Y 252.617,Z 858.479,A -85,B 0,C 180,E1 17031.849,E2 17031.849} C_VEL
LIN {X 0,Y 252.49,Z 857.28,A -85,B 0,C 180,E1 17032.096,E2 17032.096} C_VEL
LIN {X 0,Y 252.12,Z 857.28,A -85,B 0,C 180,E1 17038.712,E2 17038.712} C_VEL
LIN {X 0,Y 252.091,Z 857.941,A -85,B 0,C 180,E1 17046.355,E2 17046.355} C_VEL
LIN {X 0,Y 262.157,Z 890.693,A -85,B 0,C 180,E1 17048.907,E2 17048.907} C_VEL
LIN {X 0,Y 267.875,Z 917.312,A -85,B 0,C 180,E1 17051.885,E2 17051.885} C_VEL
LIN {X 0,Y 268.296,Z 929.032,A -85,B 0,C 180,E1 17053.42,E2 17053.42} C_VEL
LIN {X 0,Y 264.709,Z 954.181,A -85,B 0,C 180,E1 17057.455,E2 17057.455} C_VEL
LIN {X 0,Y 261.317,Z 975.378,A -85,B 0,C 180,E1 17062.603,E2 17062.603} C_VEL
LIN {X 0,Y 259.005,Z 990.682,A -85,B 0,C 180,E1 17068.322,E2 17068.322} C_VEL
LIN {X 0,Y 257.903,Z 999.868,A -85,B 0,C 180,E1 17073.937,E2 17073.937} C_VEL
LIN {X 0,Y 258.167,Z 1004.415,A -85,B 0,C 180,E1 17079.774,E2 17079.774} C_VEL
LIN {X 0,Y 258.997,Z 1004.875,A -85,B 0,C 180,E1 17083.057,E2 17083.057} C_VEL
LIN {X 0,Y 261.971,Z 1001.553,A -85,B 0,C 180,E1 17089.267,E2 17089.267} C_VEL
LIN {X 0,Y 266.776,Z 992.369,A -85,B 0,C 180,E1 17095.296,E2 17095.296} C_VEL
LIN {X 0,Y 272.905,Z 977.374,A -85,B 0,C 180,E1 17100.793,E2 17100.793} C_VEL
LIN {X 0,Y 279.45,Z 957.666,A -85,B 0,C 180,E1 17105.283,E2 17105.283} C_VEL
LIN {X 0,Y 285.121,Z 933.921,A -85,B 0,C 180,E1 17108.923,E2 17108.923} C_VEL
LIN {X 0,Y 283.91,Z 914.759,A -85,B 0,C 180,E1 17112.025,E2 17112.025} C_VEL
LIN {X 0,Y 277.706,Z 896.173,A -85,B 0,C 180,E1 17115.854,E2 17115.854} C_VEL
LIN {X 0,Y 270.293,Z 883.305,A -85,B 0,C 180,E1 17119.745,E2 17119.745} C_VEL
LIN {X 0,Y 266.6,Z 877.761,A -85,B 0,C 180,E1 17122.217,E2 17122.217} C_VEL
LIN {X 0,Y 262.973,Z 871.989,A -85,B 0,C 180,E1 17125.611,E2 17125.611} C_VEL
LIN {X 0,Y 259.75,Z 869.365,A -85,B 0,C 180,E1 17131.677,E2 17131.677} C_VEL
LIN {X 0,Y 262.782,Z 872.1,A -85,B 0,C 180,E1 17139.364,E2 17139.364} C_VEL
LIN {X 0,Y 266.657,Z 879.591,A -85,B 0,C 180,E1 17143.192,E2 17143.192} C_VEL
LIN {X 0,Y 268.991,Z 893.213,A -85,B 0,C 180,E1 17145.463,E2 17145.463} C_VEL
LIN {X 0,Y 280.809,Z 926.386,A -85,B 0,C 180,E1 17148.703,E2 17148.703} C_VEL
LIN {X 0,Y 284.207,Z 941.833,A -85,B 0,C 180,E1 17150.263,E2 17150.263} C_VEL
LIN {X 0,Y 278.046,Z 973.73,A -85,B 0,C 180,E1 17153.011,E2 17153.011} C_VEL
LIN {X 0,Y 271.208,Z 1002.633,A -85,B 0,C 180,E1 17156.904,E2 17156.904} C_VEL
LIN {X 0,Y 264.65,Z 1027.659,A -85,B 0,C 180,E1 17161.838,E2 17161.838} C_VEL
LIN {X 0,Y 259.39,Z 1049.564,A -85,B 0,C 180,E1 17168.155,E2 17168.155} C_VEL
LIN {X 0,Y 256.905,Z 1064.733,A -85,B 0,C 180,E1 17174.622,E2 17174.622} C_VEL
LIN {X 0,Y 256.464,Z 1075.019,A -85,B 0,C 180,E1 17181.514,E2 17181.514} C_VEL
LIN {X 0,Y 256.73,Z 1079.073,A -85,B 0,C 180,E1 17186.62,E2 17186.62} C_VEL
LIN {X 0,Y 257.01,Z 1080.203,A -85,B 0,C 180,E1 17190.001,E2 17190.001} C_VEL
LIN {X 0,Y 256.414,Z 1078.469,A -85,B 0,C 180,E1 17196.783,E2 17196.783} C_VEL
LIN {X 0,Y 256.319,Z 1071.822,A -85,B 0,C 180,E1 17203.668,E2 17203.668} C_VEL
LIN {X 0,Y 259.097,Z 1058.308,A -85,B 0,C 180,E1 17211.423,E2 17211.423} C_VEL
LIN {X 0,Y 265.36,Z 1039.301,A -85,B 0,C 180,E1 17218.356,E2 17218.356} C_VEL
LIN {X 0,Y 273.746,Z 1016.189,A -85,B 0,C 180,E1 17224.009,E2 17224.009} C_VEL
LIN {X 0,Y 283.045,Z 989.099,A -85,B 0,C 180,E1 17228.453,E2 17228.453} C_VEL
LIN {X 0,Y 291.92,Z 958.043,A -85,B 0,C 180,E1 17231.768,E2 17231.768} C_VEL
LIN {X 0,Y 295.063,Z 942.679,A -85,B 0,C 180,E1 17232.983,E2 17232.983} C_VEL
LIN {X 0,Y 287.953,Z 918.471,A -85,B 0,C 180,E1 17236.59,E2 17236.59} C_VEL
LIN {X 0,Y 275.536,Z 893.344,A -85,B 0,C 180,E1 17241.266,E2 17241.266} C_VEL
LIN {X 0,Y 263.662,Z 875.493,A -85,B 0,C 180,E1 17245.846,E2 17245.846} C_VEL
LIN {X 0,Y 255.848,Z 863.983,A -85,B 0,C 180,E1 17249.539,E2 17249.539} C_VEL
LIN {X 0,Y 252.405,Z 859.183,A -85,B 0,C 180,E1 17251.383,E2 17251.383} C_VEL
LIN {X 0,Y 252.202,Z 857.28,A -85,B 0,C 180,E1 17251.65,E2 17251.65} C_VEL
LIN {X 0,Y 252.223,Z 857.28,A -85,B 0,C 180,E1 17252.374,E2 17252.374} C_VEL
LIN {X 0,Y 249.734,Z 857.28,A -85,B 0,C 180,E1 17255.316,E2 17255.316} C_VEL
LIN {X 0,Y 244.625,Z 857.28,A -85,B 0,C 180,E1 17260.313,E2 17260.313} C_VEL
LIN {X 0,Y 245.416,Z 857.28,A -85,B 0,C 180,E1 17269.293,E2 17269.293} C_VEL
LIN {X 0,Y 246.216,Z 857.28,A -85,B 0,C 180,E1 17276.431,E2 17276.431} C_VEL
LIN {X 0,Y 246.602,Z 857.28,A -85,B 0,C 180,E1 17279.955,E2 17279.955} C_VEL
LIN {X 0,Y 245.58,Z 857.28,A -85,B 0,C 180,E1 17289.435,E2 17289.435} C_VEL
LIN {X 0,Y 245.191,Z 857.863,A -85,B 0,C 180,E1 17295.683,E2 17295.683} C_VEL
LIN {X 0,Y 247.605,Z 863.091,A -85,B 0,C 180,E1 17297.471,E2 17297.471} C_VEL
LIN {X 0,Y 250.222,Z 865.804,A -85,B 0,C 180,E1 17299.039,E2 17299.039} C_VEL
LIN {X 0,Y 259.98,Z 881.658,A -85,B 0,C 180,E1 17304.687,E2 17304.687} C_VEL
LIN {X 0,Y 268.981,Z 899.48,A -85,B 0,C 180,E1 17309.91,E2 17309.91} C_VEL
LIN {X 0,Y 275.75,Z 920.507,A -85,B 0,C 180,E1 17315.138,E2 17315.138} C_VEL
LIN {X 0,Y 278.776,Z 941.582,A -85,B 0,C 180,E1 17320.131,E2 17320.131} C_VEL
LIN {X 0,Y 278.447,Z 949.985,A -85,B 0,C 180,E1 17322.132,E2 17322.132} C_VEL
LIN {X 0,Y 269.393,Z 971.669,A -85,B 0,C 180,E1 17327.03,E2 17327.03} C_VEL
LIN {X 0,Y 261.639,Z 987.343,A -85,B 0,C 180,E1 17332.581,E2 17332.581} C_VEL
LIN {X 0,Y 255.582,Z 998.128,A -85,B 0,C 180,E1 17338.942,E2 17338.942} C_VEL
LIN {X 0,Y 251.952,Z 1003.428,A -85,B 0,C 180,E1 17345.123,E2 17345.123} C_VEL
LIN {X 0,Y 250.023,Z 1004.202,A -85,B 0,C 180,E1 17352.374,E2 17352.374} C_VEL
LIN {X 0,Y 250.646,Z 999.427,A -85,B 0,C 180,E1 17359.558,E2 17359.558} C_VEL
LIN {X 0,Y 253.552,Z 988.777,A -85,B 0,C 180,E1 17366.575,E2 17366.575} C_VEL
LIN {X 0,Y 258.132,Z 972.828,A -85,B 0,C 180,E1 17372.825,E2 17372.825} C_VEL
LIN {X 0,Y 263.456,Z 953.372,A -85,B 0,C 180,E1 17377.844,E2 17377.844} C_VEL
LIN {X 0,Y 267.929,Z 932.687,A -85,B 0,C 180,E1 17381.613,E2 17381.613} C_VEL
LIN {X 0,Y 264.343,Z 908.671,A -85,B 0,C 180,E1 17385.755,E2 17385.755} C_VEL
LIN {X 0,Y 256.566,Z 883.81,A -85,B 0,C 180,E1 17389.58,E2 17389.58} C_VEL
LIN {X 0,Y 244.431,Z 857.28,A -85,B 0,C 180,E1 17393.517,E2 17393.517} C_VEL
LIN {X 0,Y 244.077,Z 857.28,A -85,B 0,C 180,E1 17399.855,E2 17399.855} C_VEL
LIN {X 0,Y 244.123,Z 857.28,A -85,B 0,C 180,E1 17405.531,E2 17405.531} C_VEL
LIN {X 0,Y 254.678,Z 892.103,A -85,B 0,C 180,E1 17408.352,E2 17408.352} C_VEL
LIN {X 0,Y 260.533,Z 919.865,A -85,B 0,C 180,E1 17411.583,E2 17411.583} C_VEL
LIN {X 0,Y 260.637,Z 930.839,A -85,B 0,C 180,E1 17413.062,E2 17413.062} C_VEL
LIN {X 0,Y 256.882,Z 955.946,A -85,B 0,C 180,E1 17417.251,E2 17417.251} C_VEL
LIN {X 0,Y 253.559,Z 976.23,A -85,B 0,C 180,E1 17422.326,E2 17422.326} C_VEL
LIN {X 0,Y 251.435,Z 990.087,A -85,B 0,C 180,E1 17427.461,E2 17427.461} C_VEL
LIN {X 0,Y 250.194,Z 999.847,A -85,B 0,C 180,E1 17433.07,E2 17433.07} C_VEL
LIN {X 0,Y 250.172,Z 1005.104,A -85,B 0,C 180,E1 17438.765,E2 17438.765} C_VEL
LIN {X 0,Y 251.66,Z 1006.118,A -85,B 0,C 180,E1 17444.28,E2 17444.28} C_VEL
LIN {X 0,Y 254.501,Z 1003.057,A -85,B 0,C 180,E1 17449.768,E2 17449.768} C_VEL
LIN {X 0,Y 259.66,Z 994.042,A -85,B 0,C 180,E1 17455.968,E2 17455.968} C_VEL
LIN {X 0,Y 265.59,Z 980.82,A -85,B 0,C 180,E1 17461.118,E2 17461.118} C_VEL
LIN {X 0,Y 273.001,Z 960.748,A -85,B 0,C 180,E1 17466.007,E2 17466.007} C_VEL
LIN {X 0,Y 279.379,Z 935.817,A -85,B 0,C 180,E1 17469.991,E2 17469.991} C_VEL
LIN {X 0,Y 278.204,Z 916.367,A -85,B 0,C 180,E1 17473.389,E2 17473.389} C_VEL
LIN {X 0,Y 272.558,Z 899.32,A -85,B 0,C 180,E1 17477.33,E2 17477.33} C_VEL
LIN {X 0,Y 265.274,Z 885.924,A -85,B 0,C 180,E1 17481.978,E2 17481.978} C_VEL
LIN {X 0,Y 260.869,Z 879.495,A -85,B 0,C 180,E1 17486.086,E2 17486.086} C_VEL
LIN {X 0,Y 258.127,Z 877.201,A -85,B 0,C 180,E1 17493.288,E2 17493.288} C_VEL
LIN {X 0,Y 261.346,Z 880.772,A -85,B 0,C 180,E1 17499.694,E2 17499.694} C_VEL
LIN {X 0,Y 263.814,Z 886.385,A -85,B 0,C 180,E1 17502.352,E2 17502.352} C_VEL
LIN {X 0,Y 266.696,Z 906.414,A -85,B 0,C 180,E1 17505.661,E2 17505.661} C_VEL
LIN {X 0,Y 276.57,Z 938.859,A -85,B 0,C 180,E1 17509.131,E2 17509.131} C_VEL
LIN {X 0,Y 276.435,Z 947.29,A -85,B 0,C 180,E1 17509.874,E2 17509.874} C_VEL
LIN {X 0,Y 269.768,Z 978.654,A -85,B 0,C 180,E1 17512.891,E2 17512.891} C_VEL
LIN {X 0,Y 262.719,Z 1006.6,A -85,B 0,C 180,E1 17517.031,E2 17517.031} C_VEL
LIN {X 0,Y 256.042,Z 1031.201,A -85,B 0,C 180,E1 17522.372,E2 17522.372} C_VEL
LIN {X 0,Y 250.951,Z 1052.168,A -85,B 0,C 180,E1 17529.085,E2 17529.085} C_VEL
LIN {X 0,Y 248.801,Z 1066.485,A -85,B 0,C 180,E1 17535.913,E2 17535.913} C_VEL
LIN {X 0,Y 248.643,Z 1073.719,A -85,B 0,C 180,E1 17541.245,E2 17541.245} C_VEL
LIN {X 0,Y 248.903,Z 1077.81,A -85,B 0,C 180,E1 17546.514,E2 17546.514} C_VEL
LIN {X 0,Y 249.188,Z 1079.006,A -85,B 0,C 180,E1 17550.001,E2 17550.001} C_VEL
LIN {X 0,Y 248.554,Z 1077.339,A -85,B 0,C 180,E1 17556.999,E2 17556.999} C_VEL
LIN {X 0,Y 248.508,Z 1070.754,A -85,B 0,C 180,E1 17564.107,E2 17564.107} C_VEL
LIN {X 0,Y 251.569,Z 1057.344,A -85,B 0,C 180,E1 17572.097,E2 17572.097} C_VEL
LIN {X 0,Y 257.938,Z 1039.28,A -85,B 0,C 180,E1 17578.966,E2 17578.966} C_VEL
LIN {X 0,Y 267.198,Z 1015.299,A -85,B 0,C 180,E1 17585.012,E2 17585.012} C_VEL
LIN {X 0,Y 277.244,Z 987.258,A -85,B 0,C 180,E1 17589.665,E2 17589.665} C_VEL
LIN {X 0,Y 286.498,Z 956.1,A -85,B 0,C 180,E1 17592.97,E2 17592.97} C_VEL
LIN {X 0,Y 288.851,Z 944.917,A -85,B 0,C 180,E1 17593.893,E2 17593.893} C_VEL
LIN {X 0,Y 281.7,Z 920.382,A -85,B 0,C 180,E1 17597.821,E2 17597.821} C_VEL
LIN {X 0,Y 269.556,Z 895.295,A -85,B 0,C 180,E1 17602.905,E2 17602.905} C_VEL
LIN {X 0,Y 256.985,Z 876.57,A -85,B 0,C 180,E1 17608.321,E2 17608.321} C_VEL
LIN {X 0,Y 252.728,Z 870.581,A -85,B 0,C 180,E1 17610.502,E2 17610.502} C_VEL
LIN {X 0,Y 248.4,Z 864.193,A -85,B 0,C 180,E1 17613.011,E2 17613.011} C_VEL
LIN {X 0,Y 244.772,Z 859.517,A -85,B 0,C 180,E1 17615.404,E2 17615.404} C_VEL
LIN {X 0,Y 244.431,Z 857.28,A -85,B 0,C 180,E1 17615.976,E2 17615.976} C_VEL
LIN {X 0,Y 244.625,Z 857.28,A -85,B 0,C 180,E1 17620.313,E2 17620.313} C_VEL
LIN {X 0,Y 242.282,Z 857.28,A -85,B 0,C 180,E1 17623.352,E2 17623.352} C_VEL
LIN {X 0,Y 237.355,Z 857.28,A -85,B 0,C 180,E1 17628.518,E2 17628.518} C_VEL
LIN {X 0,Y 238.288,Z 857.28,A -85,B 0,C 180,E1 17636.312,E2 17636.312} C_VEL
LIN {X 0,Y 238.69,Z 857.28,A -85,B 0,C 180,E1 17639.954,E2 17639.954} C_VEL
LIN {X 0,Y 237.654,Z 857.28,A -85,B 0,C 180,E1 17649.753,E2 17649.753} C_VEL
LIN {X 0,Y 237.719,Z 858.391,A -85,B 0,C 180,E1 17650.508,E2 17650.508} C_VEL
LIN {X 0,Y 240.201,Z 863.371,A -85,B 0,C 180,E1 17652.924,E2 17652.924} C_VEL
LIN {X 0,Y 243.066,Z 865.992,A -85,B 0,C 180,E1 17655.066,E2 17655.066} C_VEL
LIN {X 0,Y 248.443,Z 874.679,A -85,B 0,C 180,E1 17658.95,E2 17658.95} C_VEL
LIN {X 0,Y 255.911,Z 887.068,A -85,B 0,C 180,E1 17663.711,E2 17663.711} C_VEL
LIN {X 0,Y 264.584,Z 906.006,A -85,B 0,C 180,E1 17669.513,E2 17669.513} C_VEL
LIN {X 0,Y 270.377,Z 926.775,A -85,B 0,C 180,E1 17674.932,E2 17674.932} C_VEL
LIN {X 0,Y 272.318,Z 945.931,A -85,B 0,C 180,E1 17679.745,E2 17679.745} C_VEL
LIN {X 0,Y 271.68,Z 952.855,A -85,B 0,C 180,E1 17681.434,E2 17681.434} C_VEL
LIN {X 0,Y 262.63,Z 973.277,A -85,B 0,C 180,E1 17686.225,E2 17686.225} C_VEL
LIN {X 0,Y 253.935,Z 989.82,A -85,B 0,C 180,E1 17692.372,E2 17692.372} C_VEL
LIN {X 0,Y 247.976,Z 999.67,A -85,B 0,C 180,E1 17698.611,E2 17698.611} C_VEL
LIN {X 0,Y 244.471,Z 1004.41,A -85,B 0,C 180,E1 17704.307,E2 17704.307} C_VEL
LIN {X 0,Y 242.273,Z 1005.472,A -85,B 0,C 180,E1 17711.79,E2 17711.79} C_VEL
LIN {X 0,Y 242.751,Z 1001.007,A -85,B 0,C 180,E1 17719.214,E2 17719.214} C_VEL
LIN {X 0,Y 245.641,Z 990.75,A -85,B 0,C 180,E1 17726.465,E2 17726.465} C_VEL
LIN {X 0,Y 250.41,Z 974.797,A -85,B 0,C 180,E1 17733.056,E2 17733.056} C_VEL
LIN {X 0,Y 256.21,Z 954.466,A -85,B 0,C 180,E1 17738.495,E2 17738.495} C_VEL
LIN {X 0,Y 260.786,Z 934.973,A -85,B 0,C 180,E1 17742.148,E2 17742.148} C_VEL
LIN {X 0,Y 257.419,Z 911.02,A -85,B 0,C 180,E1 17746.478,E2 17746.478} C_VEL
LIN {X 0,Y 249.981,Z 886.641,A -85,B 0,C 180,E1 17750.457,E2 17750.457} C_VEL
LIN {X 0,Y 238.095,Z 862.092,A -85,B 0,C 180,E1 17754.444,E2 17754.444} C_VEL
LIN {X 0,Y 236.423,Z 857.28,A -85,B 0,C 180,E1 17755.105,E2 17755.105} C_VEL
LIN {X 0,Y 236.175,Z 857.28,A -85,B 0,C 180,E1 17764.689,E2 17764.689} C_VEL
LIN {X 0,Y 247.22,Z 893.52,A -85,B 0,C 180,E1 17767.765,E2 17767.765} C_VEL
LIN {X 0,Y 253.048,Z 921.539,A -85,B 0,C 180,E1 17771.159,E2 17771.159} C_VEL
LIN {X 0,Y 253.045,Z 932.025,A -85,B 0,C 180,E1 17772.616,E2 17772.616} C_VEL
LIN {X 0,Y 249.169,Z 957.226,A -85,B 0,C 180,E1 17776.943,E2 17776.943} C_VEL
LIN {X 0,Y 245.591,Z 978.37,A -85,B 0,C 180,E1 17782.433,E2 17782.433} C_VEL
LIN {X 0,Y 243.305,Z 993.149,A -85,B 0,C 180,E1 17788.33,E2 17788.33} C_VEL
LIN {X 0,Y 242.176,Z 1003.428,A -85,B 0,C 180,E1 17795.235,E2 17795.235} C_VEL
LIN {X 0,Y 243.053,Z 1007.414,A -85,B 0,C 180,E1 17801.908,E2 17801.908} C_VEL
LIN {X 0,Y 244.491,Z 1007.234,A -85,B 0,C 180,E1 17805.711,E2 17805.711} C_VEL
LIN {X 0,Y 248.444,Z 1002.679,A -85,B 0,C 180,E1 17812.167,E2 17812.167} C_VEL
LIN {X 0,Y 254.398,Z 992.349,A -85,B 0,C 180,E1 17818.339,E2 17818.339} C_VEL
LIN {X 0,Y 261.679,Z 976.604,A -85,B 0,C 180,E1 17823.773,E2 17823.773} C_VEL
LIN {X 0,Y 269.467,Z 955.016,A -85,B 0,C 180,E1 17828.427,E2 17828.427} C_VEL
LIN {X 0,Y 273.869,Z 936.765,A -85,B 0,C 180,E1 17831.302,E2 17831.302} C_VEL
LIN {X 0,Y 273,Z 919.563,A -85,B 0,C 180,E1 17834.534,E2 17834.534} C_VEL
LIN {X 0,Y 267.963,Z 903.104,A -85,B 0,C 180,E1 17838.716,E2 17838.716} C_VEL
LIN {X 0,Y 261.9,Z 892.173,A -85,B 0,C 180,E1 17843.211,E2 17843.211} C_VEL
LIN {X 0,Y 259.096,Z 887.124,A -85,B 0,C 180,E1 17846.278,E2 17846.278} C_VEL
LIN {X 0,Y 256.516,Z 884.922,A -85,B 0,C 180,E1 17853.085,E2 17853.085} C_VEL
LIN {X 0,Y 259.347,Z 888.374,A -85,B 0,C 180,E1 17859.303,E2 17859.303} C_VEL
LIN {X 0,Y 261.081,Z 893.056,A -85,B 0,C 180,E1 17861.48,E2 17861.48} C_VEL
LIN {X 0,Y 264.657,Z 922.419,A -85,B 0,C 180,E1 17866.319,E2 17866.319} C_VEL
LIN {X 0,Y 270.057,Z 944.254,A -85,B 0,C 180,E1 17868.839,E2 17868.839} C_VEL
LIN {X 0,Y 263.313,Z 975.739,A -85,B 0,C 180,E1 17871.821,E2 17871.821} C_VEL
LIN {X 0,Y 255.772,Z 1004.785,A -85,B 0,C 180,E1 17876.124,E2 17876.124} C_VEL
LIN {X 0,Y 248.469,Z 1030.475,A -85,B 0,C 180,E1 17881.836,E2 17881.836} C_VEL
LIN {X 0,Y 242.988,Z 1053.052,A -85,B 0,C 180,E1 17889.237,E2 17889.237} C_VEL
LIN {X 0,Y 240.968,Z 1065.637,A -85,B 0,C 180,E1 17895.445,E2 17895.445} C_VEL
LIN {X 0,Y 240.77,Z 1072.661,A -85,B 0,C 180,E1 17900.956,E2 17900.956} C_VEL
LIN {X 0,Y 241.081,Z 1076.551,A -85,B 0,C 180,E1 17906.401,E2 17906.401} C_VEL
LIN {X 0,Y 241.39,Z 1077.812,A -85,B 0,C 180,E1 17910.001,E2 17910.001} C_VEL
LIN {X 0,Y 240.672,Z 1076.207,A -85,B 0,C 180,E1 17917.229,E2 17917.229} C_VEL
LIN {X 0,Y 240.907,Z 1068.585,A -85,B 0,C 180,E1 17925.494,E2 17925.494} C_VEL
LIN {X 0,Y 244.687,Z 1054.51,A -85,B 0,C 180,E1 17933.718,E2 17933.718} C_VEL
LIN {X 0,Y 251.961,Z 1035.677,A -85,B 0,C 180,E1 17940.717,E2 17940.717} C_VEL
LIN {X 0,Y 261.394,Z 1012.662,A -85,B 0,C 180,E1 17946.422,E2 17946.422} C_VEL
LIN {X 0,Y 271.626,Z 985.443,A -85,B 0,C 180,E1 17950.918,E2 17950.918} C_VEL
LIN {X 0,Y 281.064,Z 954.603,A -85,B 0,C 180,E1 17954.183,E2 17954.183} C_VEL
LIN {X 0,Y 282.474,Z 946.26,A -85,B 0,C 180,E1 17954.967,E2 17954.967} C_VEL
LIN {X 0,Y 275.28,Z 921.662,A -85,B 0,C 180,E1 17959.247,E2 17959.247} C_VEL
LIN {X 0,Y 263.961,Z 898.31,A -85,B 0,C 180,E1 17964.46,E2 17964.46} C_VEL
LIN {X 0,Y 251.002,Z 878.199,A -85,B 0,C 180,E1 17970.803,E2 17970.803} C_VEL
LIN {X 0,Y 245.583,Z 870.978,A -85,B 0,C 180,E1 17974.027,E2 17974.027} C_VEL
LIN {X 0,Y 241.402,Z 864.535,A -85,B 0,C 180,E1 17977.125,E2 17977.125} C_VEL
LIN {X 0,Y 237.185,Z 859.807,A -85,B 0,C 180,E1 17980.774,E2 17980.774} C_VEL
LIN {X 0,Y 236.91,Z 857.28,A -85,B 0,C 180,E1 17981.615,E2 17981.615} C_VEL
LIN {X 0,Y 237.355,Z 857.28,A -85,B 0,C 180,E1 17988.518,E2 17988.518} C_VEL
LIN {X 0,Y 235.332,Z 857.28,A -85,B 0,C 180,E1 17991.645,E2 17991.645} C_VEL
LIN {X 0,Y 230.353,Z 857.28,A -85,B 0,C 180,E1 17996.963,E2 17996.963} C_VEL
LIN {X 0,Y 230.548,Z 858.129,A -85,B 0,C 180,E1 18001.598,E2 18001.598} C_VEL
LIN {X 0,Y 233.388,Z 863.765,A -85,B 0,C 180,E1 18006.936,E2 18006.936} C_VEL
LIN {X 0,Y 235.897,Z 865.952,A -85,B 0,C 180,E1 18009.789,E2 18009.789} C_VEL
LIN {X 0,Y 239.105,Z 871.369,A -85,B 0,C 180,E1 18012.984,E2 18012.984} C_VEL
LIN {X 0,Y 241.106,Z 873.759,A -85,B 0,C 180,E1 18014.61,E2 18014.61} C_VEL
LIN {X 0,Y 248.628,Z 886.376,A -85,B 0,C 180,E1 18020.44,E2 18020.44} C_VEL
LIN {X 0,Y 256.905,Z 903.806,A -85,B 0,C 180,E1 18026.56,E2 18026.56} C_VEL
LIN {X 0,Y 263.02,Z 923.273,A -85,B 0,C 180,E1 18032.165,E2 18032.165} C_VEL
LIN {X 0,Y 265.847,Z 943.61,A -85,B 0,C 180,E1 18037.589,E2 18037.589} C_VEL
LIN {X 0,Y 265.236,Z 955.038,A -85,B 0,C 180,E1 18040.572,E2 18040.572} C_VEL
LIN {X 0,Y 256.089,Z 974.562,A -85,B 0,C 180,E1 18045.286,E2 18045.286} C_VEL
LIN {X 0,Y 247.308,Z 990.435,A -85,B 0,C 180,E1 18051.274,E2 18051.274} C_VEL
LIN {X 0,Y 240.127,Z 1001.591,A -85,B 0,C 180,E1 18058.59,E2 18058.59} C_VEL
LIN {X 0,Y 237.051,Z 1005.387,A -85,B 0,C 180,E1 18063.441,E2 18063.441} C_VEL
LIN {X 0,Y 234.556,Z 1006.724,A -85,B 0,C 180,E1 18071.169,E2 18071.169} C_VEL
LIN {X 0,Y 234.824,Z 1002.558,A -85,B 0,C 180,E1 18078.846,E2 18078.846} C_VEL
LIN {X 0,Y 237.702,Z 992.64,A -85,B 0,C 180,E1 18086.347,E2 18086.347} C_VEL
LIN {X 0,Y 242.241,Z 978.164,A -85,B 0,C 180,E1 18092.792,E2 18092.792} C_VEL
LIN {X 0,Y 248.07,Z 959.143,A -85,B 0,C 180,E1 18098.334,E2 18098.334} C_VEL
LIN {X 0,Y 253.675,Z 937.211,A -85,B 0,C 180,E1 18102.713,E2 18102.713} C_VEL
LIN {X 0,Y 250.762,Z 914.388,A -85,B 0,C 180,E1 18107.065,E2 18107.065} C_VEL
LIN {X 0,Y 243.954,Z 890.857,A -85,B 0,C 180,E1 18111.125,E2 18111.125} C_VEL
LIN {X 0,Y 232.718,Z 866.801,A -85,B 0,C 180,E1 18115.308,E2 18115.308} C_VEL
LIN {X 0,Y 228.305,Z 857.28,A -85,B 0,C 180,E1 18117.045,E2 18117.045} C_VEL
LIN {X 0,Y 228.234,Z 857.5,A -85,B 0,C 180,E1 18123.873,E2 18123.873} C_VEL
LIN {X 0,Y 239.208,Z 892.95,A -85,B 0,C 180,E1 18126.962,E2 18126.962} C_VEL
LIN {X 0,Y 245.041,Z 919.89,A -85,B 0,C 180,E1 18130.234,E2 18130.234} C_VEL
LIN {X 0,Y 245.842,Z 930.74,A -85,B 0,C 180,E1 18131.796,E2 18131.796} C_VEL
LIN {X 0,Y 241.789,Z 956.511,A -85,B 0,C 180,E1 18136.191,E2 18136.191} C_VEL
LIN {X 0,Y 238.184,Z 977.113,A -85,B 0,C 180,E1 18141.485,E2 18141.485} C_VEL
LIN {X 0,Y 235.605,Z 993.288,A -85,B 0,C 180,E1 18147.794,E2 18147.794} C_VEL
LIN {X 0,Y 234.38,Z 1003.9,A -85,B 0,C 180,E1 18154.738,E2 18154.738} C_VEL
LIN {X 0,Y 235.06,Z 1008.454,A -85,B 0,C 180,E1 18161.271,E2 18161.271} C_VEL
LIN {X 0,Y 236.461,Z 1008.836,A -85,B 0,C 180,E1 18165.215,E2 18165.215} C_VEL
LIN {X 0,Y 239.869,Z 1005.915,A -85,B 0,C 180,E1 18171.114,E2 18171.114} C_VEL
LIN {X 0,Y 245.581,Z 997.635,A -85,B 0,C 180,E1 18177.396,E2 18177.396} C_VEL
LIN {X 0,Y 252.596,Z 984.394,A -85,B 0,C 180,E1 18182.964,E2 18182.964} C_VEL
LIN {X 0,Y 260.827,Z 965.292,A -85,B 0,C 180,E1 18187.934,E2 18187.934} C_VEL
LIN {X 0,Y 268.255,Z 941.272,A -85,B 0,C 180,E1 18192.05,E2 18192.05} C_VEL
LIN {X 0,Y 268.254,Z 924.489,A -85,B 0,C 180,E1 18195.371,E2 18195.371} C_VEL
LIN {X 0,Y 264.279,Z 908.926,A -85,B 0,C 180,E1 18199.585,E2 18199.585} C_VEL
LIN {X 0,Y 259.382,Z 899.058,A -85,B 0,C 180,E1 18203.932,E2 18203.932} C_VEL
LIN {X 0,Y 257.038,Z 894.567,A -85,B 0,C 180,E1 18206.834,E2 18206.834} C_VEL
LIN {X 0,Y 254.929,Z 892.598,A -85,B 0,C 180,E1 18212.348,E2 18212.348} C_VEL
LIN {X 0,Y 257.387,Z 895.87,A -85,B 0,C 180,E1 18218.9,E2 18218.9} C_VEL
LIN {X 0,Y 258.502,Z 900.055,A -85,B 0,C 180,E1 18220.645,E2 18220.645} C_VEL
LIN {X 0,Y 262.744,Z 943.833,A -85,B 0,C 180,E1 18227.878,E2 18227.878} C_VEL
LIN {X 0,Y 256.527,Z 974.371,A -85,B 0,C 180,E1 18230.892,E2 18230.892} C_VEL
LIN {X 0,Y 249.048,Z 1003.354,A -85,B 0,C 180,E1 18235.079,E2 18235.079} C_VEL
LIN {X 0,Y 241.75,Z 1028.736,A -85,B 0,C 180,E1 18240.562,E2 18240.562} C_VEL
LIN {X 0,Y 236.031,Z 1049.811,A -85,B 0,C 180,E1 18247.365,E2 18247.365} C_VEL
LIN {X 0,Y 233.19,Z 1064.809,A -85,B 0,C 180,E1 18254.948,E2 18254.948} C_VEL
LIN {X 0,Y 232.888,Z 1071.622,A -85,B 0,C 180,E1 18260.647,E2 18260.647} C_VEL
LIN {X 0,Y 233.25,Z 1075.282,A -85,B 0,C 180,E1 18266.279,E2 18266.279} C_VEL
LIN {X 0,Y 233.592,Z 1076.606,A -85,B 0,C 180,E1 18270.001,E2 18270.001} C_VEL
LIN {X 0,Y 232.81,Z 1075.081,A -85,B 0,C 180,E1 18277.475,E2 18277.475} C_VEL
LIN {X 0,Y 233.141,Z 1067.529,A -85,B 0,C 180,E1 18286.023,E2 18286.023} C_VEL
LIN {X 0,Y 237.322,Z 1053.574,A -85,B 0,C 180,E1 18294.501,E2 18294.501} C_VEL
LIN {X 0,Y 245.017,Z 1034.87,A -85,B 0,C 180,E1 18301.687,E2 18301.687} C_VEL
LIN {X 0,Y 254.943,Z 1012.021,A -85,B 0,C 180,E1 18307.5,E2 18307.5} C_VEL
LIN {X 0,Y 265.636,Z 984.963,A -85,B 0,C 180,E1 18312.048,E2 18312.048} C_VEL
LIN {X 0,Y 275.456,Z 954.407,A -85,B 0,C 180,E1 18315.328,E2 18315.328} C_VEL
LIN {X 0,Y 276.342,Z 948.834,A -85,B 0,C 180,E1 18315.902,E2 18315.902} C_VEL
LIN {X 0,Y 269.846,Z 925.178,A -85,B 0,C 180,E1 18320.307,E2 18320.307} C_VEL
LIN {X 0,Y 259.034,Z 902.058,A -85,B 0,C 180,E1 18325.834,E2 18325.834} C_VEL
LIN {X 0,Y 248.154,Z 884.795,A -85,B 0,C 180,E1 18331.705,E2 18331.705} C_VEL
LIN {X 0,Y 242.889,Z 877.52,A -85,B 0,C 180,E1 18335.078,E2 18335.078} C_VEL
LIN {X 0,Y 239.31,Z 871.877,A -85,B 0,C 180,E1 18337.895,E2 18337.895} C_VEL
LIN {X 0,Y 235.353,Z 866.731,A -85,B 0,C 180,E1 18341.593,E2 18341.593} C_VEL
LIN {X 0,Y 234.453,Z 864.768,A -85,B 0,C 180,E1 18342.714,E2 18342.714} C_VEL
LIN {X 0,Y 229.902,Z 859.409,A -85,B 0,C 180,E1 18350.548,E2 18350.548} C_VEL
LIN {X 0,Y 229.895,Z 857.28,A -85,B 0,C 180,E1 18352.386,E2 18352.386} C_VEL
LIN {X 0,Y 230.353,Z 857.28,A -85,B 0,C 180,E1 18356.963,E2 18356.963} C_VEL
LIN {X 0,Y 230.016,Z 859.897,A -85,B 0,C 180,E1 18359.029,E2 18359.029} C_VEL
LIN {X 0,Y 229.672,Z 867.6,A -85,B 0,C 180,E1 18362.277,E2 18362.277} C_VEL
LIN {X 0,Y 234.173,Z 873.622,A -85,B 0,C 180,E1 18369.228,E2 18369.228} C_VEL
LIN {X 0,Y 237.868,Z 879.35,A -85,B 0,C 180,E1 18373.155,E2 18373.155} C_VEL
LIN {X 0,Y 245.233,Z 892.895,A -85,B 0,C 180,E1 18379.764,E2 18379.764} C_VEL
LIN {X 0,Y 253.18,Z 911.675,A -85,B 0,C 180,E1 18386.585,E2 18386.585} C_VEL
LIN {X 0,Y 258.051,Z 930.965,A -85,B 0,C 180,E1 18392.336,E2 18392.336} C_VEL
LIN {X 0,Y 259.529,Z 949.35,A -85,B 0,C 180,E1 18397.5,E2 18397.5} C_VEL
LIN {X 0,Y 258.264,Z 958.436,A -85,B 0,C 180,E1 18399.936,E2 18399.936} C_VEL
LIN {X 0,Y 248.159,Z 978.492,A -85,B 0,C 180,E1 18405.133,E2 18405.133} C_VEL
LIN {X 0,Y 238.965,Z 993.811,A -85,B 0,C 180,E1 18411.529,E2 18411.529} C_VEL
LIN {X 0,Y 232.249,Z 1003.397,A -85,B 0,C 180,E1 18418.563,E2 18418.563} C_VEL
LIN {X 0,Y 227.873,Z 1007.873,A -85,B 0,C 180,E1 18426.504,E2 18426.504} C_VEL
LIN {X 0,Y 226.487,Z 1006.732,A -85,B 0,C 180,E1 18434.489,E2 18434.489} C_VEL
LIN {X 0,Y 228.069,Z 1000.04,A -85,B 0,C 180,E1 18442.369,E2 18442.369} C_VEL
LIN {X 0,Y 232.106,Z 987.322,A -85,B 0,C 180,E1 18449.999,E2 18449.999} C_VEL
LIN {X 0,Y 237.635,Z 970.026,A -85,B 0,C 180,E1 18456.401,E2 18456.401} C_VEL
LIN {X 0,Y 244.378,Z 948.448,A -85,B 0,C 180,E1 18461.615,E2 18461.615} C_VEL
LIN {X 0,Y 246.514,Z 937.246,A -85,B 0,C 180,E1 18463.767,E2 18463.767} C_VEL
LIN {X 0,Y 243.192,Z 913.045,A -85,B 0,C 180,E1 18468.522,E2 18468.522} C_VEL
LIN {X 0,Y 235.119,Z 887.489,A -85,B 0,C 180,E1 18473.189,E2 18473.189} C_VEL
LIN {X 0,Y 222.631,Z 862.86,A -85,B 0,C 180,E1 18477.821,E2 18477.821} C_VEL
LIN {X 0,Y 220.237,Z 857.28,A -85,B 0,C 180,E1 18478.764,E2 18478.764} C_VEL
LIN {X 0,Y 220.276,Z 857.28,A -85,B 0,C 180,E1 18482.95,E2 18482.95} C_VEL
LIN {X 0,Y 231.733,Z 894.169,A -85,B 0,C 180,E1 18486.306,E2 18486.306} C_VEL
LIN {X 0,Y 237.625,Z 922.075,A -85,B 0,C 180,E1 18489.849,E2 18489.849} C_VEL
LIN {X 0,Y 238.183,Z 932.45,A -85,B 0,C 180,E1 18491.389,E2 18491.389} C_VEL
LIN {X 0,Y 234.026,Z 957.935,A -85,B 0,C 180,E1 18495.891,E2 18495.891} C_VEL
LIN {X 0,Y 230.208,Z 979.221,A -85,B 0,C 180,E1 18501.595,E2 18501.595} C_VEL
LIN {X 0,Y 227.686,Z 994.764,A -85,B 0,C 180,E1 18507.933,E2 18507.933} C_VEL
LIN {X 0,Y 226.549,Z 1005.294,A -85,B 0,C 180,E1 18515.119,E2 18515.119} C_VEL
LIN {X 0,Y 227.075,Z 1009.352,A -85,B 0,C 180,E1 18520.586,E2 18520.586} C_VEL
LIN {X 0,Y 228.417,Z 1010.242,A -85,B 0,C 180,E1 18524.682,E2 18524.682} C_VEL
LIN {X 0,Y 232.034,Z 1007.996,A -85,B 0,C 180,E1 18531.059,E2 18531.059} C_VEL
LIN {X 0,Y 237.665,Z 1000.906,A -85,B 0,C 180,E1 18537.309,E2 18537.309} C_VEL
LIN {X 0,Y 245.702,Z 987.4,A -85,B 0,C 180,E1 18543.577,E2 18543.577} C_VEL
LIN {X 0,Y 254.374,Z 969.034,A -85,B 0,C 180,E1 18548.683,E2 18548.683} C_VEL
LIN {X 0,Y 262.771,Z 945.269,A -85,B 0,C 180,E1 18552.939,E2 18552.939} C_VEL
LIN {X 0,Y 263.523,Z 929.156,A -85,B 0,C 180,E1 18556.294,E2 18556.294} C_VEL
LIN {X 0,Y 260.595,Z 914.906,A -85,B 0,C 180,E1 18560.438,E2 18560.438} C_VEL
LIN {X 0,Y 256.792,Z 905.799,A -85,B 0,C 180,E1 18564.717,E2 18564.717} C_VEL
LIN {X 0,Y 255.006,Z 901.992,A -85,B 0,C 180,E1 18567.396,E2 18567.396} C_VEL
LIN {X 0,Y 253.361,Z 900.398,A -85,B 0,C 180,E1 18573.216,E2 18573.216} C_VEL
LIN {X 0,Y 255.49,Z 903.605,A -85,B 0,C 180,E1 18578.594,E2 18578.594} C_VEL
LIN {X 0,Y 255.965,Z 906.904,A -85,B 0,C 180,E1 18579.74,E2 18579.74} C_VEL
LIN {X 0,Y 257.635,Z 947.574,A -85,B 0,C 180,E1 18586.833,E2 18586.833} C_VEL
LIN {X 0,Y 250.357,Z 979.024,A -85,B 0,C 180,E1 18590.018,E2 18590.018} C_VEL
LIN {X 0,Y 241.801,Z 1007.76,A -85,B 0,C 180,E1 18594.602,E2 18594.602} C_VEL
LIN {X 0,Y 233.82,Z 1032.257,A -85,B 0,C 180,E1 18600.508,E2 18600.508} C_VEL
LIN {X 0,Y 228.167,Z 1050.929,A -85,B 0,C 180,E1 18607.23,E2 18607.23} C_VEL
LIN {X 0,Y 225.392,Z 1064.008,A -85,B 0,C 180,E1 18614.414,E2 18614.414} C_VEL
LIN {X 0,Y 225.016,Z 1070.594,A -85,B 0,C 180,E1 18620.317,E2 18620.317} C_VEL
LIN {X 0,Y 225.441,Z 1074.018,A -85,B 0,C 180,E1 18626.15,E2 18626.15} C_VEL
LIN {X 0,Y 225.791,Z 1075.381,A -85,B 0,C 180,E1 18630.001,E2 18630.001} C_VEL
LIN {X 0,Y 224.922,Z 1073.952,A -85,B 0,C 180,E1 18637.739,E2 18637.739} C_VEL
LIN {X 0,Y 225.401,Z 1066.477,A -85,B 0,C 180,E1 18646.589,E2 18646.589} C_VEL
LIN {X 0,Y 229.966,Z 1052.64,A -85,B 0,C 180,E1 18655.339,E2 18655.339} C_VEL
LIN {X 0,Y 238.177,Z 1034.084,A -85,B 0,C 180,E1 18662.708,E2 18662.708} C_VEL
LIN {X 0,Y 248.615,Z 1011.394,A -85,B 0,C 180,E1 18668.627,E2 18668.627} C_VEL
LIN {X 0,Y 259.773,Z 984.522,A -85,B 0,C 180,E1 18673.225,E2 18673.225} C_VEL
LIN {X 0,Y 269.957,Z 954.233,A -85,B 0,C 180,E1 18676.522,E2 18676.522} C_VEL
LIN {X 0,Y 268.766,Z 943.799,A -85,B 0,C 180,E1 18678.292,E2 18678.292} C_VEL
LIN {X 0,Y 261.416,Z 921.177,A -85,B 0,C 180,E1 18683.143,E2 18683.143} C_VEL
LIN {X 0,Y 251.979,Z 902.231,A -85,B 0,C 180,E1 18688.515,E2 18688.515} C_VEL
LIN {X 0,Y 242.006,Z 885.901,A -85,B 0,C 180,E1 18694.88,E2 18694.88} C_VEL
LIN {X 0,Y 237.007,Z 878.923,A -85,B 0,C 180,E1 18698.9,E2 18698.9} C_VEL
LIN {X 0,Y 233.455,Z 873.146,A -85,B 0,C 180,E1 18702.625,E2 18702.625} C_VEL
LIN {X 0,Y 228.683,Z 866.384,A -85,B 0,C 180,E1 18711.512,E2 18711.512} C_VEL
LIN {X 0,Y 228.647,Z 865.081,A -85,B 0,C 180,E1 18712.344,E2 18712.344} C_VEL
LIN {X 0,Y 229.314,Z 865.725,A -85,B 0,C 180,E1 18721.015,E2 18721.015} C_VEL
LIN {X 0,Y 229.672,Z 867.6,A -85,B 0,C 180,E1 18722.277,E2 18722.277} C_VEL
LIN {X 0,Y 233.117,Z 883.588,A -85,B 0,C 180,E1 18730.013,E2 18730.013} C_VEL
LIN {X 0,Y 236.534,Z 889.038,A -85,B 0,C 180,E1 18733.849,E2 18733.849} C_VEL
LIN {X 0,Y 241.755,Z 899.563,A -85,B 0,C 180,E1 18739.14,E2 18739.14} C_VEL
LIN {X 0,Y 248.377,Z 916.895,A -85,B 0,C 180,E1 18745.767,E2 18745.767} C_VEL
LIN {X 0,Y 252.523,Z 936.676,A -85,B 0,C 180,E1 18751.999,E2 18751.999} C_VEL
LIN {X 0,Y 253.048,Z 954.821,A -85,B 0,C 180,E1 18757.384,E2 18757.384} C_VEL
LIN {X 0,Y 251.771,Z 960.905,A -85,B 0,C 180,E1 18759.055,E2 18759.055} C_VEL
LIN {X 0,Y 241.187,Z 980.626,A -85,B 0,C 180,E1 18764.391,E2 18764.391} C_VEL
LIN {X 0,Y 231.739,Z 995.454,A -85,B 0,C 180,E1 18770.88,E2 18770.88} C_VEL
LIN {X 0,Y 225.219,Z 1004.236,A -85,B 0,C 180,E1 18777.463,E2 18777.463} C_VEL
LIN {X 0,Y 220.379,Z 1008.992,A -85,B 0,C 180,E1 18785.654,E2 18785.654} C_VEL
LIN {X 0,Y 218.666,Z 1008.135,A -85,B 0,C 180,E1 18793.919,E2 18793.919} C_VEL
LIN {X 0,Y 220.11,Z 1001.746,A -85,B 0,C 180,E1 18802.091,E2 18802.091} C_VEL
LIN {X 0,Y 224.17,Z 989.375,A -85,B 0,C 180,E1 18809.999,E2 18809.999} C_VEL
LIN {X 0,Y 229.909,Z 972.374,A -85,B 0,C 180,E1 18816.662,E2 18816.662} C_VEL
LIN {X 0,Y 237.076,Z 950.515,A -85,B 0,C 180,E1 18822.212,E2 18822.212} C_VEL
LIN {X 0,Y 239.456,Z 939.47,A -85,B 0,C 180,E1 18824.415,E2 18824.415} C_VEL
LIN {X 0,Y 236.597,Z 916.22,A -85,B 0,C 180,E1 18829.237,E2 18829.237} C_VEL
LIN {X 0,Y 229.809,Z 893.276,A -85,B 0,C 180,E1 18833.666,E2 18833.666} C_VEL
LIN {X 0,Y 217.81,Z 868.311,A -85,B 0,C 180,E1 18838.707,E2 18838.707} C_VEL
LIN {X 0,Y 212.376,Z 858.582,A -85,B 0,C 180,E1 18840.722,E2 18840.722} C_VEL
LIN {X 0,Y 212.29,Z 857.28,A -85,B 0,C 180,E1 18840.902,E2 18840.902} C_VEL
LIN {X 0,Y 212.363,Z 857.453,A -85,B 0,C 180,E1 18842.048,E2 18842.048} C_VEL
LIN {X 0,Y 224.118,Z 894.929,A -85,B 0,C 180,E1 18845.575,E2 18845.575} C_VEL
LIN {X 0,Y 229.955,Z 922.297,A -85,B 0,C 180,E1 18849.143,E2 18849.143} C_VEL
LIN {X 0,Y 230.406,Z 934.951,A -85,B 0,C 180,E1 18851.08,E2 18851.08} C_VEL
LIN {X 0,Y 226.184,Z 960.011,A -85,B 0,C 180,E1 18855.726,E2 18855.726} C_VEL
LIN {X 0,Y 222.362,Z 980.618,A -85,B 0,C 180,E1 18861.487,E2 18861.487} C_VEL
LIN {X 0,Y 219.84,Z 995.63,A -85,B 0,C 180,E1 18867.797,E2 18867.797} C_VEL
LIN {X 0,Y 218.729,Z 1005.209,A -85,B 0,C 180,E1 18874.139,E2 18874.139} C_VEL
LIN {X 0,Y 219.087,Z 1010.054,A -85,B 0,C 180,E1 18879.848,E2 18879.848} C_VEL
LIN {X 0,Y 220.369,Z 1011.517,A -85,B 0,C 180,E1 18884.127,E2 18884.127} C_VEL
LIN {X 0,Y 224.105,Z 1010.041,A -85,B 0,C 180,E1 18890.915,E2 18890.915} C_VEL
LIN {X 0,Y 230.766,Z 1002.658,A -85,B 0,C 180,E1 18898.169,E2 18898.169} C_VEL
LIN {X 0,Y 239.349,Z 989.456,A -85,B 0,C 180,E1 18904.58,E2 18904.58} C_VEL
LIN {X 0,Y 248.59,Z 971.528,A -85,B 0,C 180,E1 18909.767,E2 18909.767} C_VEL
LIN {X 0,Y 257.784,Z 947.291,A -85,B 0,C 180,E1 18914.276,E2 18914.276} C_VEL
LIN {X 0,Y 258.887,Z 932.775,A -85,B 0,C 180,E1 18917.517,E2 18917.517} C_VEL
LIN {X 0,Y 256.833,Z 920.337,A -85,B 0,C 180,E1 18921.497,E2 18921.497} C_VEL
LIN {X 0,Y 254.08,Z 912.428,A -85,B 0,C 180,E1 18925.588,E2 18925.588} C_VEL
LIN {X 0,Y 252.858,Z 909.46,A -85,B 0,C 180,E1 18928.03,E2 18928.03} C_VEL
LIN {X 0,Y 251.897,Z 908.341,A -85,B 0,C 180,E1 18934.143,E2 18934.143} C_VEL
LIN {X 0,Y 253.541,Z 911.122,A -85,B 0,C 180,E1 18938.171,E2 18938.171} C_VEL
LIN {X 0,Y 253.268,Z 949.802,A -85,B 0,C 180,E1 18945.365,E2 18945.365} C_VEL
LIN {X 0,Y 244.706,Z 982.015,A -85,B 0,C 180,E1 18948.899,E2 18948.899} C_VEL
LIN {X 0,Y 235.492,Z 1009.073,A -85,B 0,C 180,E1 18953.503,E2 18953.503} C_VEL
LIN {X 0,Y 226.784,Z 1032.919,A -85,B 0,C 180,E1 18959.624,E2 18959.624} C_VEL
LIN {X 0,Y 220.376,Z 1051.651,A -85,B 0,C 180,E1 18966.933,E2 18966.933} C_VEL
LIN {X 0,Y 217.404,Z 1064.502,A -85,B 0,C 180,E1 18974.863,E2 18974.863} C_VEL
LIN {X 0,Y 217.246,Z 1070.834,A -85,B 0,C 180,E1 18981.989,E2 18981.989} C_VEL
LIN {X 0,Y 217.989,Z 1074.149,A -85,B 0,C 180,E1 18990.001,E2 18990.001} C_VEL
LIN {X 0,Y 217.062,Z 1072.831,A -85,B 0,C 180,E1 18998.021,E2 18998.021} C_VEL
LIN {X 0,Y 217.657,Z 1065.423,A -85,B 0,C 180,E1 19007.197,E2 19007.197} C_VEL
LIN {X 0,Y 222.635,Z 1051.719,A -85,B 0,C 180,E1 19016.236,E2 19016.236} C_VEL
LIN {X 0,Y 231.389,Z 1033.303,A -85,B 0,C 180,E1 19023.794,E2 19023.794} C_VEL
LIN {X 0,Y 242.362,Z 1010.802,A -85,B 0,C 180,E1 19029.818,E2 19029.818} C_VEL
LIN {X 0,Y 254.436,Z 983.074,A -85,B 0,C 180,E1 19034.6,E2 19034.6} C_VEL
LIN {X 0,Y 264.121,Z 953.64,A -85,B 0,C 180,E1 19037.95,E2 19037.95} C_VEL
LIN {X 0,Y 259.376,Z 933.734,A -85,B 0,C 180,E1 19042.164,E2 19042.164} C_VEL
LIN {X 0,Y 250.85,Z 913.16,A -85,B 0,C 180,E1 19047.729,E2 19047.729} C_VEL
LIN {X 0,Y 242.143,Z 897.517,A -85,B 0,C 180,E1 19053.564,E2 19053.564} C_VEL
LIN {X 0,Y 235.423,Z 886.501,A -85,B 0,C 180,E1 19059.244,E2 19059.244} C_VEL
LIN {X 0,Y 231.067,Z 879.863,A -85,B 0,C 180,E1 19064.275,E2 19064.275} C_VEL
LIN {X 0,Y 227.583,Z 873.73,A -85,B 0,C 180,E1 19072.188,E2 19072.188} C_VEL
LIN {X 0,Y 228.116,Z 873.249,A -85,B 0,C 180,E1 19080.427,E2 19080.427} C_VEL
LIN {X 0,Y 230.794,Z 879.289,A -85,B 0,C 180,E1 19086.6,E2 19086.6} C_VEL
LIN {X 0,Y 232.409,Z 881.547,A -85,B 0,C 180,E1 19088.918,E2 19088.918} C_VEL
LIN {X 0,Y 233.117,Z 883.588,A -85,B 0,C 180,E1 19090.013,E2 19090.013} C_VEL
LIN {X 0,Y 234.753,Z 890.246,A -85,B 0,C 180,E1 19092.762,E2 19092.762} C_VEL
LIN {X 0,Y 236.886,Z 903.222,A -85,B 0,C 180,E1 19097.102,E2 19097.102} C_VEL
LIN {X 0,Y 242.672,Z 919.096,A -85,B 0,C 180,E1 19103.864,E2 19103.864} C_VEL
LIN {X 0,Y 246.352,Z 937.219,A -85,B 0,C 180,E1 19110.059,E2 19110.059} C_VEL
LIN {X 0,Y 246.95,Z 955.135,A -85,B 0,C 180,E1 19115.706,E2 19115.706} C_VEL
LIN {X 0,Y 245.716,Z 962.61,A -85,B 0,C 180,E1 19117.962,E2 19117.962} C_VEL
LIN {X 0,Y 235.158,Z 981.351,A -85,B 0,C 180,E1 19123.111,E2 19123.111} C_VEL
LIN {X 0,Y 224.779,Z 996.781,A -85,B 0,C 180,E1 19129.996,E2 19129.996} C_VEL
LIN {X 0,Y 218.268,Z 1005.045,A -85,B 0,C 180,E1 19136.292,E2 19136.292} C_VEL
LIN {X 0,Y 212.917,Z 1010.102,A -85,B 0,C 180,E1 19144.742,E2 19144.742} C_VEL
LIN {X 0,Y 210.884,Z 1009.517,A -85,B 0,C 180,E1 19153.309,E2 19153.309} C_VEL
LIN {X 0,Y 212.177,Z 1003.431,A -85,B 0,C 180,E1 19161.793,E2 19161.793} C_VEL
LIN {X 0,Y 216.221,Z 991.438,A -85,B 0,C 180,E1 19169.999,E2 19169.999} C_VEL
LIN {X 0,Y 222.316,Z 974.38,A -85,B 0,C 180,E1 19177.054,E2 19177.054} C_VEL
LIN {X 0,Y 229.718,Z 952.621,A -85,B 0,C 180,E1 19182.851,E2 19182.851} C_VEL
LIN {X 0,Y 232.428,Z 941.698,A -85,B 0,C 180,E1 19185.102,E2 19185.102} C_VEL
LIN {X 0,Y 229.942,Z 919.137,A -85,B 0,C 180,E1 19190.02,E2 19190.02} C_VEL
LIN {X 0,Y 223.089,Z 895.285,A -85,B 0,C 180,E1 19194.908,E2 19194.908} C_VEL
LIN {X 0,Y 211.939,Z 872.01,A -85,B 0,C 180,E1 19200.003,E2 19200.003} C_VEL
LIN {X 0,Y 207.984,Z 866.642,A -85,B 0,C 180,E1 19201.524,E2 19201.524} C_VEL
LIN {X 0,Y 207.323,Z 866.604,A -85,B 0,C 180,E1 19201.875,E2 19201.875} C_VEL
LIN {X 0,Y 217.253,Z 898.686,A -85,B 0,C 180,E1 19205.163,E2 19205.163} C_VEL
LIN {X 0,Y 222.815,Z 926.349,A -85,B 0,C 180,E1 19209.011,E2 19209.011} C_VEL
LIN {X 0,Y 222.658,Z 936.921,A -85,B 0,C 180,E1 19210.68,E2 19210.68} C_VEL
LIN {X 0,Y 218.386,Z 961.449,A -85,B 0,C 180,E1 19215.43,E2 19215.43} C_VEL
LIN {X 0,Y 214.367,Z 982.719,A -85,B 0,C 180,E1 19221.643,E2 19221.643} C_VEL
LIN {X 0,Y 211.851,Z 997.753,A -85,B 0,C 180,E1 19228.357,E2 19228.357} C_VEL
LIN {X 0,Y 210.864,Z 1007.77,A -85,B 0,C 180,E1 19235.685,E2 19235.685} C_VEL
LIN {X 0,Y 212.297,Z 1012.634,A -85,B 0,C 180,E1 19243.487,E2 19243.487} C_VEL
LIN {X 0,Y 215.44,Z 1012.402,A -85,B 0,C 180,E1 19249.697,E2 19249.697} C_VEL
LIN {X 0,Y 221.716,Z 1007.01,A -85,B 0,C 180,E1 19257.116,E2 19257.116} C_VEL
LIN {X 0,Y 230.289,Z 995.941,A -85,B 0,C 180,E1 19263.816,E2 19263.816} C_VEL
LIN {X 0,Y 240.48,Z 978.917,A -85,B 0,C 180,E1 19269.678,E2 19269.678} C_VEL
LIN {X 0,Y 250.403,Z 957.357,A -85,B 0,C 180,E1 19274.259,E2 19274.259} C_VEL
LIN {X 0,Y 253.74,Z 945.611,A -85,B 0,C 180,E1 19276.504,E2 19276.504} C_VEL
LIN {X 0,Y 254.223,Z 933.332,A -85,B 0,C 180,E1 19279.759,E2 19279.759} C_VEL
LIN {X 0,Y 252.358,Z 921.95,A -85,B 0,C 180,E1 19284.412,E2 19284.412} C_VEL
LIN {X 0,Y 250.808,Z 917.058,A -85,B 0,C 180,E1 19288.115,E2 19288.115} C_VEL
LIN {X 0,Y 250.184,Z 916.109,A -85,B 0,C 180,E1 19294.202,E2 19294.202} C_VEL
LIN {X 0,Y 251.439,Z 917.915,A -85,B 0,C 180,E1 19297.38,E2 19297.38} C_VEL
LIN {X 0,Y 248.736,Z 954.52,A -85,B 0,C 180,E1 19304.194,E2 19304.194} C_VEL
LIN {X 0,Y 239.121,Z 984.89,A -85,B 0,C 180,E1 19307.721,E2 19307.721} C_VEL
LIN {X 0,Y 228.836,Z 1011.636,A -85,B 0,C 180,E1 19312.605,E2 19312.605} C_VEL
LIN {X 0,Y 218.966,Z 1035.508,A -85,B 0,C 180,E1 19319.351,E2 19319.351} C_VEL
LIN {X 0,Y 212.457,Z 1052.737,A -85,B 0,C 180,E1 19326.84,E2 19326.84} C_VEL
LIN {X 0,Y 209.419,Z 1064.797,A -85,B 0,C 180,E1 19335.344,E2 19335.344} C_VEL
LIN {X 0,Y 209.358,Z 1069.691,A -85,B 0,C 180,E1 19341.685,E2 19341.685} C_VEL
LIN {X 0,Y 210.19,Z 1072.916,A -85,B 0,C 180,E1 19350.001,E2 19350.001} C_VEL
LIN {X 0,Y 209.17,Z 1071.695,A -85,B 0,C 180,E1 19358.325,E2 19358.325} C_VEL
LIN {X 0,Y 209.942,Z 1064.382,A -85,B 0,C 180,E1 19367.85,E2 19367.85} C_VEL
LIN {X 0,Y 215.4,Z 1050.805,A -85,B 0,C 180,E1 19377.188,E2 19377.188} C_VEL
LIN {X 0,Y 224.699,Z 1032.551,A -85,B 0,C 180,E1 19384.944,E2 19384.944} C_VEL
LIN {X 0,Y 236.241,Z 1010.195,A -85,B 0,C 180,E1 19391.068,E2 19391.068} C_VEL
LIN {X 0,Y 248.25,Z 984.069,A -85,B 0,C 180,E1 19395.69,E2 19395.69} C_VEL
LIN {X 0,Y 258.138,Z 956.377,A -85,B 0,C 180,E1 19398.977,E2 19398.977} C_VEL
LIN {X 0,Y 253.245,Z 935.383,A -85,B 0,C 180,E1 19403.779,E2 19403.779} C_VEL
LIN {X 0,Y 245.415,Z 915.871,A -85,B 0,C 180,E1 19409.582,E2 19409.582} C_VEL
LIN {X 0,Y 237.08,Z 900.02,A -85,B 0,C 180,E1 19416.203,E2 19416.203} C_VEL
LIN {X 0,Y 232.854,Z 893.376,A -85,B 0,C 180,E1 19420.262,E2 19420.262} C_VEL
LIN {X 0,Y 229.38,Z 887.391,A -85,B 0,C 180,E1 19424.892,E2 19424.892} C_VEL
LIN {X 0,Y 226.386,Z 881.044,A -85,B 0,C 180,E1 19432.87,E2 19432.87} C_VEL
LIN {X 0,Y 226.81,Z 881.386,A -85,B 0,C 180,E1 19440.31,E2 19440.31} C_VEL
LIN {X 0,Y 229.619,Z 887.395,A -85,B 0,C 180,E1 19447.229,E2 19447.229} C_VEL
LIN {X 0,Y 234.156,Z 897.073,A -85,B 0,C 180,E1 19453.836,E2 19453.836} C_VEL
LIN {X 0,Y 236.886,Z 903.222,A -85,B 0,C 180,E1 19457.102,E2 19457.102} C_VEL
LIN {X 0,Y 238.067,Z 910.992,A -85,B 0,C 180,E1 19459.637,E2 19459.637} C_VEL
LIN {X 0,Y 238.259,Z 925.915,A -85,B 0,C 180,E1 19463.614,E2 19463.614} C_VEL
LIN {X 0,Y 240.891,Z 944.156,A -85,B 0,C 180,E1 19470.119,E2 19470.119} C_VEL
LIN {X 0,Y 240.256,Z 961.62,A -85,B 0,C 180,E1 19475.938,E2 19475.938} C_VEL
LIN {X 0,Y 238.484,Z 966.589,A -85,B 0,C 180,E1 19477.331,E2 19477.331} C_VEL
LIN {X 0,Y 227.252,Z 985.163,A -85,B 0,C 180,E1 19482.87,E2 19482.87} C_VEL
LIN {X 0,Y 216.389,Z 999.948,A -85,B 0,C 180,E1 19490.214,E2 19490.214} C_VEL
LIN {X 0,Y 209.497,Z 1007.815,A -85,B 0,C 180,E1 19497.298,E2 19497.298} C_VEL
LIN {X 0,Y 205.514,Z 1011.156,A -85,B 0,C 180,E1 19503.765,E2 19503.765} C_VEL
LIN {X 0,Y 203.116,Z 1010.842,A -85,B 0,C 180,E1 19512.651,E2 19512.651} C_VEL
LIN {X 0,Y 204.203,Z 1005.057,A -85,B 0,C 180,E1 19521.471,E2 19521.471} C_VEL
LIN {X 0,Y 208.294,Z 993.446,A -85,B 0,C 180,E1 19529.999,E2 19529.999} C_VEL
LIN {X 0,Y 214.604,Z 976.574,A -85,B 0,C 180,E1 19537.418,E2 19537.418} C_VEL
LIN {X 0,Y 222.359,Z 954.741,A -85,B 0,C 180,E1 19543.535,E2 19543.535} C_VEL
LIN {X 0,Y 225.388,Z 943.659,A -85,B 0,C 180,E1 19545.899,E2 19545.899} C_VEL
LIN {X 0,Y 223.227,Z 921.619,A -85,B 0,C 180,E1 19550.926,E2 19550.926} C_VEL
LIN {X 0,Y 216.769,Z 898.333,A -85,B 0,C 180,E1 19556.02,E2 19556.02} C_VEL
LIN {X 0,Y 207.717,Z 878.302,A -85,B 0,C 180,E1 19560.678,E2 19560.678} C_VEL
LIN {X 0,Y 203.431,Z 878.374,A -85,B 0,C 180,E1 19562.023,E2 19562.023} C_VEL
LIN {X 0,Y 211.352,Z 906.542,A -85,B 0,C 180,E1 19565.279,E2 19565.279} C_VEL
LIN {X 0,Y 215.903,Z 933.155,A -85,B 0,C 180,E1 19569.383,E2 19569.383} C_VEL
LIN {X 0,Y 211.234,Z 959.494,A -85,B 0,C 180,E1 19574.312,E2 19574.312} C_VEL
LIN {X 0,Y 207.014,Z 981.378,A -85,B 0,C 180,E1 19580.565,E2 19580.565} C_VEL
LIN {X 0,Y 204.095,Z 997.945,A -85,B 0,C 180,E1 19587.869,E2 19587.869} C_VEL
LIN {X 0,Y 203.017,Z 1008.842,A -85,B 0,C 180,E1 19595.855,E2 19595.855} C_VEL
LIN {X 0,Y 204.682,Z 1013.952,A -85,B 0,C 180,E1 19604.073,E2 19604.073} C_VEL
LIN {X 0,Y 208.998,Z 1013.438,A -85,B 0,C 180,E1 19611.726,E2 19611.726} C_VEL
LIN {X 0,Y 215.978,Z 1007.595,A -85,B 0,C 180,E1 19619.048,E2 19619.048} C_VEL
LIN {X 0,Y 225.447,Z 995.991,A -85,B 0,C 180,E1 19625.829,E2 19625.829} C_VEL
LIN {X 0,Y 236.366,Z 978.687,A -85,B 0,C 180,E1 19631.59,E2 19631.59} C_VEL
LIN {X 0,Y 246.843,Z 957.064,A -85,B 0,C 180,E1 19636.062,E2 19636.062} C_VEL
LIN {X 0,Y 249.678,Z 945.641,A -85,B 0,C 180,E1 19638.603,E2 19638.603} C_VEL
LIN {X 0,Y 249.888,Z 934.143,A -85,B 0,C 180,E1 19642.39,E2 19642.39} C_VEL
LIN {X 0,Y 248.695,Z 926.45,A -85,B 0,C 180,E1 19646.698,E2 19646.698} C_VEL
LIN {X 0,Y 247.933,Z 923.745,A -85,B 0,C 180,E1 19650.346,E2 19650.346} C_VEL
LIN {X 0,Y 248.893,Z 924.762,A -85,B 0,C 180,E1 19656.271,E2 19656.271} C_VEL
LIN {X 0,Y 244.373,Z 958.172,A -85,B 0,C 180,E1 19662.825,E2 19662.825} C_VEL
LIN {X 0,Y 234.149,Z 986.47,A -85,B 0,C 180,E1 19666.286,E2 19666.286} C_VEL
LIN {X 0,Y 222.716,Z 1012.961,A -85,B 0,C 180,E1 19671.392,E2 19671.392} C_VEL
LIN {X 0,Y 212.086,Z 1035.895,A -85,B 0,C 180,E1 19678.294,E2 19678.294} C_VEL
LIN {X 0,Y 204.973,Z 1052.433,A -85,B 0,C 180,E1 19686.031,E2 19686.031} C_VEL
LIN {X 0,Y 201.645,Z 1063.918,A -85,B 0,C 180,E1 19694.765,E2 19694.765} C_VEL
LIN {X 0,Y 201.502,Z 1068.562,A -85,B 0,C 180,E1 19701.358,E2 19701.358} C_VEL
LIN {X 0,Y 202.382,Z 1071.683,A -85,B 0,C 180,E1 19710.002,E2 19710.002} C_VEL
LIN {X 0,Y 201.311,Z 1070.547,A -85,B 0,C 180,E1 19718.653,E2 19718.653} C_VEL
LIN {X 0,Y 202.276,Z 1063.358,A -85,B 0,C 180,E1 19728.537,E2 19728.537} C_VEL
LIN {X 0,Y 208.156,Z 1050.047,A -85,B 0,C 180,E1 19738.131,E2 19738.131} C_VEL
LIN {X 0,Y 218.1,Z 1031.799,A -85,B 0,C 180,E1 19746.164,E2 19746.164} C_VEL
LIN {X 0,Y 230.24,Z 1009.625,A -85,B 0,C 180,E1 19752.382,E2 19752.382} C_VEL
LIN {X 0,Y 242.911,Z 983.33,A -85,B 0,C 180,E1 19757.095,E2 19757.095} C_VEL
LIN {X 0,Y 252.111,Z 958.819,A -85,B 0,C 180,E1 19760.098,E2 19760.098} C_VEL
LIN {X 0,Y 247.615,Z 938.235,A -85,B 0,C 180,E1 19765.188,E2 19765.188} C_VEL
LIN {X 0,Y 240.912,Z 920.75,A -85,B 0,C 180,E1 19770.814,E2 19770.814} C_VEL
LIN {X 0,Y 233.984,Z 906.577,A -85,B 0,C 180,E1 19777.113,E2 19777.113} C_VEL
LIN {X 0,Y 230.213,Z 900.281,A -85,B 0,C 180,E1 19781.166,E2 19781.166} C_VEL
LIN {X 0,Y 227.567,Z 894.99,A -85,B 0,C 180,E1 19785.262,E2 19785.262} C_VEL
LIN {X 0,Y 224.85,Z 888.393,A -85,B 0,C 180,E1 19794.156,E2 19794.156} C_VEL
LIN {X 0,Y 225.193,Z 889.181,A -85,B 0,C 180,E1 19800.071,E2 19800.071} C_VEL
LIN {X 0,Y 227.902,Z 896.505,A -85,B 0,C 180,E1 19808.023,E2 19808.023} C_VEL
LIN {X 0,Y 232.725,Z 908.018,A -85,B 0,C 180,E1 19815.593,E2 19815.593} C_VEL
LIN {X 0,Y 237.803,Z 924.051,A -85,B 0,C 180,E1 19822.892,E2 19822.892} C_VEL
LIN {X 0,Y 238.259,Z 925.915,A -85,B 0,C 180,E1 19823.614,E2 19823.614} C_VEL
LIN {X 0,Y 238.076,Z 934.508,A -85,B 0,C 180,E1 19826.008,E2 19826.008} C_VEL
LIN {X 0,Y 235.15,Z 949.873,A -85,B 0,C 180,E1 19829.838,E2 19829.838} C_VEL
LIN {X 0,Y 233.623,Z 966.239,A -85,B 0,C 180,E1 19835.605,E2 19835.605} C_VEL
LIN {X 0,Y 221.693,Z 985.463,A -85,B 0,C 180,E1 19841.298,E2 19841.298} C_VEL
LIN {X 0,Y 210.086,Z 1000.594,A -85,B 0,C 180,E1 19848.767,E2 19848.767} C_VEL
LIN {X 0,Y 202.244,Z 1008.986,A -85,B 0,C 180,E1 19856.42,E2 19856.42} C_VEL
LIN {X 0,Y 198.145,Z 1012.216,A -85,B 0,C 180,E1 19862.71,E2 19862.71} C_VEL
LIN {X 0,Y 195.373,Z 1012.166,A -85,B 0,C 180,E1 19871.94,E2 19871.94} C_VEL
LIN {X 0,Y 196.228,Z 1006.682,A -85,B 0,C 180,E1 19881.121,E2 19881.121} C_VEL
LIN {X 0,Y 200.351,Z 995.399,A -85,B 0,C 180,E1 19889.998,E2 19889.998} C_VEL
LIN {X 0,Y 206.997,Z 978.518,A -85,B 0,C 180,E1 19897.861,E2 19897.861} C_VEL
LIN {X 0,Y 215.038,Z 956.81,A -85,B 0,C 180,E1 19904.265,E2 19904.265} C_VEL
LIN {X 0,Y 218.371,Z 945.526,A -85,B 0,C 180,E1 19906.748,E2 19906.748} C_VEL
LIN {X 0,Y 216.455,Z 923.407,A -85,B 0,C 180,E1 19912.041,E2 19912.041} C_VEL
LIN {X 0,Y 210.402,Z 901.035,A -85,B 0,C 180,E1 19917.251,E2 19917.251} C_VEL
LIN {X 0,Y 204.591,Z 887.587,A -85,B 0,C 180,E1 19920.627,E2 19920.627} C_VEL
LIN {X 0,Y 200.658,Z 889.908,A -85,B 0,C 180,E1 19921.546,E2 19921.546} C_VEL
LIN {X 0,Y 198.953,Z 889.175,A -85,B 0,C 180,E1 19922.187,E2 19922.187} C_VEL
LIN {X 0,Y 205.955,Z 917.815,A -85,B 0,C 180,E1 19926.022,E2 19926.022} C_VEL
LIN {X 0,Y 207.973,Z 936.376,A -85,B 0,C 180,E1 19929.108,E2 19929.108} C_VEL
LIN {X 0,Y 203.106,Z 962.649,A -85,B 0,C 180,E1 19934.376,E2 19934.376} C_VEL
LIN {X 0,Y 198.898,Z 983.798,A -85,B 0,C 180,E1 19940.859,E2 19940.859} C_VEL
LIN {X 0,Y 196.132,Z 999.428,A -85,B 0,C 180,E1 19948.118,E2 19948.118} C_VEL
LIN {X 0,Y 195.163,Z 1009.938,A -85,B 0,C 180,E1 19956.087,E2 19956.087} C_VEL
LIN {X 0,Y 196.115,Z 1014.263,A -85,B 0,C 180,E1 19962.08,E2 19962.08} C_VEL
LIN {X 0,Y 199.888,Z 1015.605,A -85,B 0,C 180,E1 19969.957,E2 19969.957} C_VEL
LIN {X 0,Y 206.979,Z 1011.425,A -85,B 0,C 180,E1 19978.126,E2 19978.126} C_VEL
LIN {X 0,Y 216.218,Z 1002.031,A -85,B 0,C 180,E1 19985.071,E2 19985.071} C_VEL
LIN {X 0,Y 226.862,Z 987.84,A -85,B 0,C 180,E1 19990.922,E2 19990.922} C_VEL
LIN {X 0,Y 238.345,Z 968.053,A -85,B 0,C 180,E1 19995.941,E2 19995.941} C_VEL
LIN {X 0,Y 244.175,Z 954.526,A -85,B 0,C 180,E1 19998.556,E2 19998.556} C_VEL
LIN {X 0,Y 246.07,Z 942.913,A -85,B 0,C 180,E1 20002.05,E2 20002.05} C_VEL
LIN {X 0,Y 245.821,Z 934.331,A -85,B 0,C 180,E1 20006.496,E2 20006.496} C_VEL
LIN {X 0,Y 245.43,Z 931.266,A -85,B 0,C 180,E1 20010.271,E2 20010.271} C_VEL
LIN {X 0,Y 246.277,Z 931.962,A -85,B 0,C 180,E1 20015.5,E2 20015.5} C_VEL
LIN {X 0,Y 240.532,Z 960.599,A -85,B 0,C 180,E1 20021.281,E2 20021.281} C_VEL
LIN {X 0,Y 228.818,Z 989.397,A -85,B 0,C 180,E1 20024.995,E2 20024.995} C_VEL
LIN {X 0,Y 216.213,Z 1015.242,A -85,B 0,C 180,E1 20030.351,E2 20030.351} C_VEL
LIN {X 0,Y 204.749,Z 1037.343,A -85,B 0,C 180,E1 20037.582,E2 20037.582} C_VEL
LIN {X 0,Y 196.9,Z 1053.742,A -85,B 0,C 180,E1 20046.192,E2 20046.192} C_VEL
LIN {X 0,Y 193.847,Z 1063.03,A -85,B 0,C 180,E1 20054.136,E2 20054.136} C_VEL
LIN {X 0,Y 193.631,Z 1067.376,A -85,B 0,C 180,E1 20061.004,E2 20061.004} C_VEL
LIN {X 0,Y 194.578,Z 1070.445,A -85,B 0,C 180,E1 20070.002,E2 20070.002} C_VEL
LIN {X 0,Y 193.429,Z 1069.39,A -85,B 0,C 180,E1 20079.008,E2 20079.008} C_VEL
LIN {X 0,Y 194.871,Z 1061.721,A -85,B 0,C 180,E1 20089.911,E2 20089.911} C_VEL
LIN {X 0,Y 201.496,Z 1048.387,A -85,B 0,C 180,E1 20099.655,E2 20099.655} C_VEL
LIN {X 0,Y 212.78,Z 1029.198,A -85,B 0,C 180,E1 20108.103,E2 20108.103} C_VEL
LIN {X 0,Y 226.413,Z 1005.25,A -85,B 0,C 180,E1 20114.602,E2 20114.602} C_VEL
LIN {X 0,Y 239.928,Z 977.743,A -85,B 0,C 180,E1 20119.226,E2 20119.226} C_VEL
LIN {X 0,Y 246.174,Z 961.836,A -85,B 0,C 180,E1 20121.133,E2 20121.133} C_VEL
LIN {X 0,Y 242.528,Z 942.902,A -85,B 0,C 180,E1 20126.112,E2 20126.112} C_VEL
LIN {X 0,Y 236.288,Z 924.962,A -85,B 0,C 180,E1 20132.244,E2 20132.244} C_VEL
LIN {X 0,Y 228.965,Z 908.924,A -85,B 0,C 180,E1 20140.243,E2 20140.243} C_VEL
LIN {X 0,Y 225.153,Z 902.237,A -85,B 0,C 180,E1 20146.09,E2 20146.09} C_VEL
LIN {X 0,Y 223.129,Z 896.074,A -85,B 0,C 180,E1 20154.111,E2 20154.111} C_VEL
LIN {X 0,Y 223.256,Z 896.773,A -85,B 0,C 180,E1 20159.708,E2 20159.708} C_VEL
LIN {X 0,Y 225.299,Z 903.968,A -85,B 0,C 180,E1 20167.671,E2 20167.671} C_VEL
LIN {X 0,Y 228.809,Z 913.198,A -85,B 0,C 180,E1 20174.311,E2 20174.311} C_VEL
LIN {X 0,Y 232.931,Z 929.131,A -85,B 0,C 180,E1 20181.961,E2 20181.961} C_VEL
LIN {X 0,Y 235.051,Z 945.624,A -85,B 0,C 180,E1 20188.316,E2 20188.316} C_VEL
LIN {X 0,Y 235.15,Z 949.873,A -85,B 0,C 180,E1 20189.838,E2 20189.838} C_VEL
LIN {X 0,Y 233.115,Z 958.418,A -85,B 0,C 180,E1 20192.239,E2 20192.239} C_VEL
LIN {X 0,Y 224.492,Z 973.6,A -85,B 0,C 180,E1 20195.819,E2 20195.819} C_VEL
LIN {X 0,Y 211.734,Z 991.801,A -85,B 0,C 180,E1 20202.123,E2 20202.123} C_VEL
LIN {X 0,Y 201.295,Z 1004.045,A -85,B 0,C 180,E1 20209.266,E2 20209.266} C_VEL
LIN {X 0,Y 193.937,Z 1011.087,A -85,B 0,C 180,E1 20216.871,E2 20216.871} C_VEL
LIN {X 0,Y 188.763,Z 1014.062,A -85,B 0,C 180,E1 20226.354,E2 20226.354} C_VEL
LIN {X 0,Y 187.45,Z 1011.583,A -85,B 0,C 180,E1 20235.975,E2 20235.975} C_VEL
LIN {X 0,Y 190.03,Z 1003.548,A -85,B 0,C 180,E1 20245.428,E2 20245.428} C_VEL
LIN {X 0,Y 195.26,Z 990.471,A -85,B 0,C 180,E1 20253.889,E2 20253.889} C_VEL
LIN {X 0,Y 202.652,Z 972.05,A -85,B 0,C 180,E1 20261.309,E2 20261.309} C_VEL
LIN {X 0,Y 211.288,Z 949.107,A -85,B 0,C 180,E1 20267.192,E2 20267.192} C_VEL
LIN {X 0,Y 210.06,Z 927.273,A -85,B 0,C 180,E1 20272.739,E2 20272.739} C_VEL
LIN {X 0,Y 204.906,Z 906.056,A -85,B 0,C 180,E1 20277.988,E2 20277.988} C_VEL
LIN {X 0,Y 201.455,Z 897.013,A -85,B 0,C 180,E1 20280.348,E2 20280.348} C_VEL
LIN {X 0,Y 195.571,Z 899.979,A -85,B 0,C 180,E1 20281.762,E2 20281.762} C_VEL
LIN {X 0,Y 194.102,Z 899.797,A -85,B 0,C 180,E1 20282.495,E2 20282.495} C_VEL
LIN {X 0,Y 199.744,Z 926.904,A -85,B 0,C 180,E1 20286.649,E2 20286.649} C_VEL
LIN {X 0,Y 200.373,Z 937.636,A -85,B 0,C 180,E1 20288.545,E2 20288.545} C_VEL
LIN {X 0,Y 195.338,Z 963.917,A -85,B 0,C 180,E1 20294.002,E2 20294.002} C_VEL
LIN {X 0,Y 191.025,Z 985.093,A -85,B 0,C 180,E1 20300.743,E2 20300.743} C_VEL
LIN {X 0,Y 188.288,Z 1000.129,A -85,B 0,C 180,E1 20307.964,E2 20307.964} C_VEL
LIN {X 0,Y 187.322,Z 1010.919,A -85,B 0,C 180,E1 20316.239,E2 20316.239} C_VEL
LIN {X 0,Y 188.947,Z 1016.162,A -85,B 0,C 180,E1 20324.062,E2 20324.062} C_VEL
LIN {X 0,Y 192.699,Z 1017.031,A -85,B 0,C 180,E1 20331.021,E2 20331.021} C_VEL
LIN {X 0,Y 199.127,Z 1013.911,A -85,B 0,C 180,E1 20338.258,E2 20338.258} C_VEL
LIN {X 0,Y 208.412,Z 1005.845,A -85,B 0,C 180,E1 20345.261,E2 20345.261} C_VEL
LIN {X 0,Y 219.929,Z 992.315,A -85,B 0,C 180,E1 20351.547,E2 20351.547} C_VEL
LIN {X 0,Y 232.41,Z 973.204,A -85,B 0,C 180,E1 20356.833,E2 20356.833} C_VEL
LIN {X 0,Y 239.784,Z 958.245,A -85,B 0,C 180,E1 20359.841,E2 20359.841} C_VEL
LIN {X 0,Y 242.065,Z 948.247,A -85,B 0,C 180,E1 20363.064,E2 20363.064} C_VEL
LIN {X 0,Y 242.547,Z 941.122,A -85,B 0,C 180,E1 20367.05,E2 20367.05} C_VEL
LIN {X 0,Y 242.616,Z 938.744,A -85,B 0,C 180,E1 20369.989,E2 20369.989} C_VEL
LIN {X 0,Y 243.129,Z 939.69,A -85,B 0,C 180,E1 20374.794,E2 20374.794} C_VEL
LIN {X 0,Y 236.482,Z 964.151,A -85,B 0,C 180,E1 20379.801,E2 20379.801} C_VEL
LIN {X 0,Y 223.577,Z 992.211,A -85,B 0,C 180,E1 20383.636,E2 20383.636} C_VEL
LIN {X 0,Y 210.39,Z 1016.423,A -85,B 0,C 180,E1 20388.954,E2 20388.954} C_VEL
LIN {X 0,Y 198.045,Z 1037.562,A -85,B 0,C 180,E1 20396.341,E2 20396.341} C_VEL
LIN {X 0,Y 189.502,Z 1053.282,A -85,B 0,C 180,E1 20405.201,E2 20405.201} C_VEL
LIN {X 0,Y 186.095,Z 1062.086,A -85,B 0,C 180,E1 20413.457,E2 20413.457} C_VEL
LIN {X 0,Y 185.761,Z 1066.16,A -85,B 0,C 180,E1 20420.62,E2 20420.62} C_VEL
LIN {X 0,Y 186.762,Z 1069.208,A -85,B 0,C 180,E1 20430.002,E2 20430.002} C_VEL
LIN {X 0,Y 185.563,Z 1068.236,A -85,B 0,C 180,E1 20439.394,E2 20439.394} C_VEL
LIN {X 0,Y 187.198,Z 1060.845,A -85,B 0,C 180,E1 20450.592,E2 20450.592} C_VEL
LIN {X 0,Y 194.082,Z 1048.179,A -85,B 0,C 180,E1 20460.449,E2 20460.449} C_VEL
LIN {X 0,Y 205.342,Z 1030.325,A -85,B 0,C 180,E1 20468.846,E2 20468.846} C_VEL
LIN {X 0,Y 219.713,Z 1006.686,A -85,B 0,C 180,E1 20475.642,E2 20475.642} C_VEL
LIN {X 0,Y 233.552,Z 980.102,A -85,B 0,C 180,E1 20480.341,E2 20480.341} C_VEL
LIN {X 0,Y 240.248,Z 964.642,A -85,B 0,C 180,E1 20482.245,E2 20482.245} C_VEL
LIN {X 0,Y 236.994,Z 945.719,A -85,B 0,C 180,E1 20487.62,E2 20487.62} C_VEL
LIN {X 0,Y 231.299,Z 928.841,A -85,B 0,C 180,E1 20494,E2 20494} C_VEL
LIN {X 0,Y 226.25,Z 916.715,A -85,B 0,C 180,E1 20500.408,E2 20500.408} C_VEL
LIN {X 0,Y 222.728,Z 909.583,A -85,B 0,C 180,E1 20506.493,E2 20506.493} C_VEL
LIN {X 0,Y 221.069,Z 903.793,A -85,B 0,C 180,E1 20514.056,E2 20514.056} C_VEL
LIN {X 0,Y 221.003,Z 904.437,A -85,B 0,C 180,E1 20519.459,E2 20519.459} C_VEL
LIN {X 0,Y 222.538,Z 911.892,A -85,B 0,C 180,E1 20527.767,E2 20527.767} C_VEL
LIN {X 0,Y 225.383,Z 921.378,A -85,B 0,C 180,E1 20534.534,E2 20534.534} C_VEL
LIN {X 0,Y 228.198,Z 934.934,A -85,B 0,C 180,E1 20541.343,E2 20541.343} C_VEL
LIN {X 0,Y 229.379,Z 951.27,A -85,B 0,C 180,E1 20547.969,E2 20547.969} C_VEL
LIN {X 0,Y 227.729,Z 967.174,A -85,B 0,C 180,E1 20553.949,E2 20553.949} C_VEL
LIN {X 0,Y 224.492,Z 973.6,A -85,B 0,C 180,E1 20555.819,E2 20555.819} C_VEL
LIN {X 0,Y 214.594,Z 984.554,A -85,B 0,C 180,E1 20558.314,E2 20558.314} C_VEL
LIN {X 0,Y 205.638,Z 993.01,A -85,B 0,C 180,E1 20560.804,E2 20560.804} C_VEL
LIN {X 0,Y 204.72,Z 994.037,A -85,B 0,C 180,E1 20561.274,E2 20561.274} C_VEL
LIN {X 0,Y 193.62,Z 1006.146,A -85,B 0,C 180,E1 20568.87,E2 20568.87} C_VEL
LIN {X 0,Y 187.057,Z 1012.017,A -85,B 0,C 180,E1 20575.485,E2 20575.485} C_VEL
LIN {X 0,Y 181.294,Z 1015.257,A -85,B 0,C 180,E1 20585.317,E2 20585.317} C_VEL
LIN {X 0,Y 179.599,Z 1013.052,A -85,B 0,C 180,E1 20595.348,E2 20595.348} C_VEL
LIN {X 0,Y 182.048,Z 1005.315,A -85,B 0,C 180,E1 20605.228,E2 20605.228} C_VEL
LIN {X 0,Y 187.4,Z 992.578,A -85,B 0,C 180,E1 20614.052,E2 20614.052} C_VEL
LIN {X 0,Y 194.962,Z 974.634,A -85,B 0,C 180,E1 20621.761,E2 20621.761} C_VEL
LIN {X 0,Y 203.698,Z 952.863,A -85,B 0,C 180,E1 20627.72,E2 20627.72} C_VEL
LIN {X 0,Y 204.31,Z 938.654,A -85,B 0,C 180,E1 20631.475,E2 20631.475} C_VEL
LIN {X 0,Y 201.256,Z 918.151,A -85,B 0,C 180,E1 20636.831,E2 20636.831} C_VEL
LIN {X 0,Y 197.182,Z 906.482,A -85,B 0,C 180,E1 20640.182,E2 20640.182} C_VEL
LIN {X 0,Y 189.845,Z 909.175,A -85,B 0,C 180,E1 20642.082,E2 20642.082} C_VEL
LIN {X 0,Y 188.642,Z 909,A -85,B 0,C 180,E1 20642.789,E2 20642.789} C_VEL
LIN {X 0,Y 193.258,Z 935.867,A -85,B 0,C 180,E1 20647.424,E2 20647.424} C_VEL
LIN {X 0,Y 188.129,Z 962.4,A -85,B 0,C 180,E1 20652.884,E2 20652.884} C_VEL
LIN {X 0,Y 183.673,Z 983.566,A -85,B 0,C 180,E1 20659.522,E2 20659.522} C_VEL
LIN {X 0,Y 180.462,Z 1000.55,A -85,B 0,C 180,E1 20667.652,E2 20667.652} C_VEL
LIN {X 0,Y 179.483,Z 1012.143,A -85,B 0,C 180,E1 20676.707,E2 20676.707} C_VEL
LIN {X 0,Y 181.708,Z 1017.73,A -85,B 0,C 180,E1 20685.593,E2 20685.593} C_VEL
LIN {X 0,Y 184.504,Z 1018.565,A -85,B 0,C 180,E1 20690.619,E2 20690.619} C_VEL
LIN {X 0,Y 191.286,Z 1016.252,A -85,B 0,C 180,E1 20698.411,E2 20698.411} C_VEL
LIN {X 0,Y 202.232,Z 1007.992,A -85,B 0,C 180,E1 20706.5,E2 20706.5} C_VEL
LIN {X 0,Y 215.305,Z 993.897,A -85,B 0,C 180,E1 20713.25,E2 20713.25} C_VEL
LIN {X 0,Y 228.275,Z 975.492,A -85,B 0,C 180,E1 20718.407,E2 20718.407} C_VEL
LIN {X 0,Y 235.662,Z 961.873,A -85,B 0,C 180,E1 20721.227,E2 20721.227} C_VEL
LIN {X 0,Y 238.392,Z 952.263,A -85,B 0,C 180,E1 20724.756,E2 20724.756} C_VEL
LIN {X 0,Y 239.128,Z 947.891,A -85,B 0,C 180,E1 20727.574,E2 20727.574} C_VEL
LIN {X 0,Y 239.577,Z 945.989,A -85,B 0,C 180,E1 20732.265,E2 20732.265} C_VEL
LIN {X 0,Y 240.019,Z 946.051,A -85,B 0,C 180,E1 20733.723,E2 20733.723} C_VEL
LIN {X 0,Y 232.588,Z 967.647,A -85,B 0,C 180,E1 20738.264,E2 20738.264} C_VEL
LIN {X 0,Y 218.476,Z 994.942,A -85,B 0,C 180,E1 20742.214,E2 20742.214} C_VEL
LIN {X 0,Y 203.567,Z 1019.336,A -85,B 0,C 180,E1 20747.982,E2 20747.982} C_VEL
LIN {X 0,Y 189.985,Z 1040.053,A -85,B 0,C 180,E1 20756.094,E2 20756.094} C_VEL
LIN {X 0,Y 181.378,Z 1054.256,A -85,B 0,C 180,E1 20765.332,E2 20765.332} C_VEL
LIN {X 0,Y 177.918,Z 1062.779,A -85,B 0,C 180,E1 20775.21,E2 20775.21} C_VEL
LIN {X 0,Y 178.359,Z 1066.208,A -85,B 0,C 180,E1 20785.132,E2 20785.132} C_VEL
LIN {X 0,Y 178.927,Z 1067.964,A -85,B 0,C 180,E1 20790.002,E2 20790.002} C_VEL
LIN {X 0,Y 177.695,Z 1067.081,A -85,B 0,C 180,E1 20799.814,E2 20799.814} C_VEL
LIN {X 0,Y 179.412,Z 1060.331,A -85,B 0,C 180,E1 20810.94,E2 20810.94} C_VEL
LIN {X 0,Y 187.096,Z 1047.314,A -85,B 0,C 180,E1 20821.714,E2 20821.714} C_VEL
LIN {X 0,Y 199.221,Z 1029.468,A -85,B 0,C 180,E1 20830.355,E2 20830.355} C_VEL
LIN {X 0,Y 213.896,Z 1006.594,A -85,B 0,C 180,E1 20837.066,E2 20837.066} C_VEL
LIN {X 0,Y 228.556,Z 979.766,A -85,B 0,C 180,E1 20841.877,E2 20841.877} C_VEL
LIN {X 0,Y 234.297,Z 966.825,A -85,B 0,C 180,E1 20843.575,E2 20843.575} C_VEL
LIN {X 0,Y 231.492,Z 948.768,A -85,B 0,C 180,E1 20849.132,E2 20849.132} C_VEL
LIN {X 0,Y 226.877,Z 933.735,A -85,B 0,C 180,E1 20855.306,E2 20855.306} C_VEL
LIN {X 0,Y 222.27,Z 922.264,A -85,B 0,C 180,E1 20862.107,E2 20862.107} C_VEL
LIN {X 0,Y 220.727,Z 918.018,A -85,B 0,C 180,E1 20865.413,E2 20865.413} C_VEL
LIN {X 0,Y 218.54,Z 911.194,A -85,B 0,C 180,E1 20875.978,E2 20875.978} C_VEL
LIN {X 0,Y 218.247,Z 914.425,A -85,B 0,C 180,E1 20881.936,E2 20881.936} C_VEL
LIN {X 0,Y 219.324,Z 918.329,A -85,B 0,C 180,E1 20886.885,E2 20886.885} C_VEL
LIN {X 0,Y 221.351,Z 927.514,A -85,B 0,C 180,E1 20893.794,E2 20893.794} C_VEL
LIN {X 0,Y 223.391,Z 941.314,A -85,B 0,C 180,E1 20901.033,E2 20901.033} C_VEL
LIN {X 0,Y 223.532,Z 956.565,A -85,B 0,C 180,E1 20907.545,E2 20907.545} C_VEL
LIN {X 0,Y 221.395,Z 970.472,A -85,B 0,C 180,E1 20913.092,E2 20913.092} C_VEL
LIN {X 0,Y 209.132,Z 988.594,A -85,B 0,C 180,E1 20918.896,E2 20918.896} C_VEL
LIN {X 0,Y 204.72,Z 994.037,A -85,B 0,C 180,E1 20921.274,E2 20921.274} C_VEL
LIN {X 0,Y 194.908,Z 1002.102,A -85,B 0,C 180,E1 20924.76,E2 20924.76} C_VEL
LIN {X 0,Y 186.348,Z 1007.908,A -85,B 0,C 180,E1 20928.169,E2 20928.169} C_VEL
LIN {X 0,Y 185.571,Z 1008.571,A -85,B 0,C 180,E1 20928.762,E2 20928.762} C_VEL
LIN {X 0,Y 176.691,Z 1015.308,A -85,B 0,C 180,E1 20938.809,E2 20938.809} C_VEL
LIN {X 0,Y 172.282,Z 1016.124,A -85,B 0,C 180,E1 20949.417,E2 20949.417} C_VEL
LIN {X 0,Y 172.374,Z 1011.458,A -85,B 0,C 180,E1 20959.88,E2 20959.88} C_VEL
LIN {X 0,Y 176.546,Z 1001.138,A -85,B 0,C 180,E1 20969.998,E2 20969.998} C_VEL
LIN {X 0,Y 183.574,Z 985.658,A -85,B 0,C 180,E1 20978.792,E2 20978.792} C_VEL
LIN {X 0,Y 192.283,Z 965.476,A -85,B 0,C 180,E1 20985.996,E2 20985.996} C_VEL
LIN {X 0,Y 197.638,Z 951.203,A -85,B 0,C 180,E1 20989.581,E2 20989.581} C_VEL
LIN {X 0,Y 196.574,Z 930.029,A -85,B 0,C 180,E1 20995.569,E2 20995.569} C_VEL
LIN {X 0,Y 193.563,Z 915.261,A -85,B 0,C 180,E1 20999.683,E2 20999.683} C_VEL
LIN {X 0,Y 183.409,Z 917.664,A -85,B 0,C 180,E1 21002.605,E2 21002.605} C_VEL
LIN {X 0,Y 182.684,Z 917.501,A -85,B 0,C 180,E1 21003.121,E2 21003.121} C_VEL
LIN {X 0,Y 185.304,Z 939.264,A -85,B 0,C 180,E1 21007.145,E2 21007.145} C_VEL
LIN {X 0,Y 179.989,Z 965.508,A -85,B 0,C 180,E1 21012.967,E2 21012.967} C_VEL
LIN {X 0,Y 175.291,Z 987.025,A -85,B 0,C 180,E1 21020.295,E2 21020.295} C_VEL
LIN {X 0,Y 172.409,Z 1002.49,A -85,B 0,C 180,E1 21028.294,E2 21028.294} C_VEL
LIN {X 0,Y 171.65,Z 1013.086,A -85,B 0,C 180,E1 21036.947,E2 21036.947} C_VEL
LIN {X 0,Y 173.511,Z 1018.438,A -85,B 0,C 180,E1 21044.897,E2 21044.897} C_VEL
LIN {X 0,Y 176.282,Z 1019.917,A -85,B 0,C 180,E1 21050.177,E2 21050.177} C_VEL
LIN {X 0,Y 181.914,Z 1019.101,A -85,B 0,C 180,E1 21057.117,E2 21057.117} C_VEL
LIN {X 0,Y 192.667,Z 1012.872,A -85,B 0,C 180,E1 21065.693,E2 21065.693} C_VEL
LIN {X 0,Y 205.787,Z 1001.204,A -85,B 0,C 180,E1 21072.801,E2 21072.801} C_VEL
LIN {X 0,Y 220.198,Z 983.916,A -85,B 0,C 180,E1 21078.588,E2 21078.588} C_VEL
LIN {X 0,Y 231.577,Z 965.811,A -85,B 0,C 180,E1 21082.58,E2 21082.58} C_VEL
LIN {X 0,Y 234.66,Z 957.433,A -85,B 0,C 180,E1 21086.031,E2 21086.031} C_VEL
LIN {X 0,Y 235.461,Z 954.646,A -85,B 0,C 180,E1 21088.041,E2 21088.041} C_VEL
LIN {X 0,Y 236.355,Z 953.16,A -85,B 0,C 180,E1 21092.759,E2 21092.759} C_VEL
LIN {X 0,Y 229.525,Z 969.815,A -85,B 0,C 180,E1 21096.542,E2 21096.542} C_VEL
LIN {X 0,Y 214.123,Z 996.638,A -85,B 0,C 180,E1 21100.526,E2 21100.526} C_VEL
LIN {X 0,Y 197.845,Z 1020.539,A -85,B 0,C 180,E1 21106.47,E2 21106.47} C_VEL
LIN {X 0,Y 183.404,Z 1040.246,A -85,B 0,C 180,E1 21114.701,E2 21114.701} C_VEL
LIN {X 0,Y 174.028,Z 1053.71,A -85,B 0,C 180,E1 21124.216,E2 21124.216} C_VEL
LIN {X 0,Y 170.134,Z 1061.712,A -85,B 0,C 180,E1 21134.517,E2 21134.517} C_VEL
LIN {X 0,Y 170.508,Z 1064.877,A -85,B 0,C 180,E1 21144.907,E2 21144.907} C_VEL
LIN {X 0,Y 171.105,Z 1066.723,A -85,B 0,C 180,E1 21150.002,E2 21150.002} C_VEL
LIN {X 0,Y 169.836,Z 1065.928,A -85,B 0,C 180,E1 21160.272,E2 21160.272} C_VEL
LIN {X 0,Y 171.851,Z 1059.317,A -85,B 0,C 180,E1 21171.908,E2 21171.908} C_VEL
LIN {X 0,Y 180.008,Z 1046.772,A -85,B 0,C 180,E1 21182.873,E2 21182.873} C_VEL
LIN {X 0,Y 193.132,Z 1028.731,A -85,B 0,C 180,E1 21191.908,E2 21191.908} C_VEL
LIN {X 0,Y 208.767,Z 1005.607,A -85,B 0,C 180,E1 21198.794,E2 21198.794} C_VEL
LIN {X 0,Y 223.743,Z 979.534,A -85,B 0,C 180,E1 21203.476,E2 21203.476} C_VEL
LIN {X 0,Y 228.15,Z 970.499,A -85,B 0,C 180,E1 21204.664,E2 21204.664} C_VEL
LIN {X 0,Y 226.872,Z 956.146,A -85,B 0,C 180,E1 21209.154,E2 21209.154} C_VEL
LIN {X 0,Y 222.833,Z 940.097,A -85,B 0,C 180,E1 21215.897,E2 21215.897} C_VEL
LIN {X 0,Y 218.92,Z 929.112,A -85,B 0,C 180,E1 21222.654,E2 21222.654} C_VEL
LIN {X 0,Y 216.587,Z 923.639,A -85,B 0,C 180,E1 21228.157,E2 21228.157} C_VEL
LIN {X 0,Y 215.837,Z 918.66,A -85,B 0,C 180,E1 21235.928,E2 21235.928} C_VEL
LIN {X 0,Y 215.513,Z 923.152,A -85,B 0,C 180,E1 21243.975,E2 21243.975} C_VEL
LIN {X 0,Y 217.045,Z 931.998,A -85,B 0,C 180,E1 21252.022,E2 21252.022} C_VEL
LIN {X 0,Y 218.272,Z 945.487,A -85,B 0,C 180,E1 21259.714,E2 21259.714} C_VEL
LIN {X 0,Y 217.905,Z 959.444,A -85,B 0,C 180,E1 21266.125,E2 21266.125} C_VEL
LIN {X 0,Y 214.921,Z 974.07,A -85,B 0,C 180,E1 21272.285,E2 21272.285} C_VEL
LIN {X 0,Y 201.033,Z 992.574,A -85,B 0,C 180,E1 21278.609,E2 21278.609} C_VEL
LIN {X 0,Y 188.898,Z 1005.454,A -85,B 0,C 180,E1 21286.058,E2 21286.058} C_VEL
LIN {X 0,Y 185.571,Z 1008.571,A -85,B 0,C 180,E1 21288.762,E2 21288.762} C_VEL
LIN {X 0,Y 176.929,Z 1013.559,A -85,B 0,C 180,E1 21293.324,E2 21293.324} C_VEL
LIN {X 0,Y 168.984,Z 1016.575,A -85,B 0,C 180,E1 21298.413,E2 21298.413} C_VEL
LIN {X 0,Y 164.672,Z 1017.381,A -85,B 0,C 180,E1 21308.419,E2 21308.419} C_VEL
LIN {X 0,Y 164.422,Z 1012.995,A -85,B 0,C 180,E1 21319.385,E2 21319.385} C_VEL
LIN {X 0,Y 168.607,Z 1002.971,A -85,B 0,C 180,E1 21329.998,E2 21329.998} C_VEL
LIN {X 0,Y 175.725,Z 987.893,A -85,B 0,C 180,E1 21339.188,E2 21339.188} C_VEL
LIN {X 0,Y 184.844,Z 968.174,A -85,B 0,C 180,E1 21346.658,E2 21346.658} C_VEL
LIN {X 0,Y 190.829,Z 953.166,A -85,B 0,C 180,E1 21350.645,E2 21350.645} C_VEL
LIN {X 0,Y 190.274,Z 933.828,A -85,B 0,C 180,E1 21356.421,E2 21356.421} C_VEL
LIN {X 0,Y 188.781,Z 923.91,A -85,B 0,C 180,E1 21359.319,E2 21359.319} C_VEL
LIN {X 0,Y 187.782,Z 923.175,A -85,B 0,C 180,E1 21359.822,E2 21359.822} C_VEL
LIN {X 0,Y 177.766,Z 925.811,A -85,B 0,C 180,E1 21362.7,E2 21362.7} C_VEL
LIN {X 0,Y 176.405,Z 925.193,A -85,B 0,C 180,E1 21363.462,E2 21363.462} C_VEL
LIN {X 0,Y 177.82,Z 939.841,A -85,B 0,C 180,E1 21366.353,E2 21366.353} C_VEL
LIN {X 0,Y 172.289,Z 966.335,A -85,B 0,C 180,E1 21372.414,E2 21372.414} C_VEL
LIN {X 0,Y 167.452,Z 987.791,A -85,B 0,C 180,E1 21379.99,E2 21379.99} C_VEL
LIN {X 0,Y 164.462,Z 1003.676,A -85,B 0,C 180,E1 21388.53,E2 21388.53} C_VEL
LIN {X 0,Y 163.936,Z 1015.021,A -85,B 0,C 180,E1 21398.402,E2 21398.402} C_VEL
LIN {X 0,Y 166.507,Z 1020.212,A -85,B 0,C 180,E1 21406.934,E2 21406.934} C_VEL
LIN {X 0,Y 171.918,Z 1021.366,A -85,B 0,C 180,E1 21415.014,E2 21415.014} C_VEL
LIN {X 0,Y 182.17,Z 1017.594,A -85,B 0,C 180,E1 21424.188,E2 21424.188} C_VEL
LIN {X 0,Y 195.757,Z 1007.935,A -85,B 0,C 180,E1 21432.119,E2 21432.119} C_VEL
LIN {X 0,Y 210.729,Z 993.067,A -85,B 0,C 180,E1 21438.368,E2 21438.368} C_VEL
LIN {X 0,Y 225.658,Z 973.212,A -85,B 0,C 180,E1 21443.206,E2 21443.206} C_VEL
LIN {X 0,Y 229.249,Z 966.771,A -85,B 0,C 180,E1 21445.094,E2 21445.094} C_VEL
LIN {X 0,Y 231.029,Z 962.664,A -85,B 0,C 180,E1 21447.348,E2 21447.348} C_VEL
LIN {X 0,Y 232.415,Z 960.053,A -85,B 0,C 180,E1 21451.451,E2 21451.451} C_VEL
LIN {X 0,Y 232.33,Z 960.461,A -85,B 0,C 180,E1 21452.094,E2 21452.094} C_VEL
LIN {X 0,Y 226.089,Z 973.091,A -85,B 0,C 180,E1 21454.895,E2 21454.895} C_VEL
LIN {X 0,Y 209.326,Z 999.29,A -85,B 0,C 180,E1 21458.965,E2 21458.965} C_VEL
LIN {X 0,Y 192.26,Z 1021.757,A -85,B 0,C 180,E1 21464.868,E2 21464.868} C_VEL
LIN {X 0,Y 176.072,Z 1041.389,A -85,B 0,C 180,E1 21473.801,E2 21473.801} C_VEL
LIN {X 0,Y 166.019,Z 1054.197,A -85,B 0,C 180,E1 21484.126,E2 21484.126} C_VEL
LIN {X 0,Y 162.395,Z 1060.6,A -85,B 0,C 180,E1 21493.759,E2 21493.759} C_VEL
LIN {X 0,Y 162.66,Z 1063.535,A -85,B 0,C 180,E1 21504.661,E2 21504.661} C_VEL
LIN {X 0,Y 163.272,Z 1065.479,A -85,B 0,C 180,E1 21510.002,E2 21510.002} C_VEL
LIN {X 0,Y 161.972,Z 1064.775,A -85,B 0,C 180,E1 21520.777,E2 21520.777} C_VEL
LIN {X 0,Y 164.231,Z 1058.545,A -85,B 0,C 180,E1 21532.676,E2 21532.676} C_VEL
LIN {X 0,Y 172.746,Z 1046.485,A -85,B 0,C 180,E1 21543.902,E2 21543.902} C_VEL
LIN {X 0,Y 186.239,Z 1029.226,A -85,B 0,C 180,E1 21553.058,E2 21553.058} C_VEL
LIN {X 0,Y 202.343,Z 1006.984,A -85,B 0,C 180,E1 21560.044,E2 21560.044} C_VEL
LIN {X 0,Y 218.423,Z 980.579,A -85,B 0,C 180,E1 21564.97,E2 21564.97} C_VEL
LIN {X 0,Y 222.401,Z 972.912,A -85,B 0,C 180,E1 21566.003,E2 21566.003} C_VEL
LIN {X 0,Y 221.124,Z 957.612,A -85,B 0,C 180,E1 21571.316,E2 21571.316} C_VEL
LIN {X 0,Y 217.998,Z 944.532,A -85,B 0,C 180,E1 21577.469,E2 21577.469} C_VEL
LIN {X 0,Y 214.685,Z 934.248,A -85,B 0,C 180,E1 21584.618,E2 21584.618} C_VEL
LIN {X 0,Y 212.765,Z 926.392,A -85,B 0,C 180,E1 21595.063,E2 21595.063} C_VEL
LIN {X 0,Y 212.046,Z 928.805,A -85,B 0,C 180,E1 21601.467,E2 21601.467} C_VEL
LIN {X 0,Y 212.427,Z 934.463,A -85,B 0,C 180,E1 21608.139,E2 21608.139} C_VEL
LIN {X 0,Y 213.062,Z 942.747,A -85,B 0,C 180,E1 21614.342,E2 21614.342} C_VEL
LIN {X 0,Y 212.978,Z 956.474,A -85,B 0,C 180,E1 21621.849,E2 21621.849} C_VEL
LIN {X 0,Y 210.776,Z 970.434,A -85,B 0,C 180,E1 21628.323,E2 21628.323} C_VEL
LIN {X 0,Y 208.15,Z 977.73,A -85,B 0,C 180,E1 21631.402,E2 21631.402} C_VEL
LIN {X 0,Y 193.879,Z 995.274,A -85,B 0,C 180,E1 21637.746,E2 21637.746} C_VEL
LIN {X 0,Y 180.902,Z 1008.045,A -85,B 0,C 180,E1 21645.805,E2 21645.805} C_VEL
LIN {X 0,Y 171.456,Z 1015.289,A -85,B 0,C 180,E1 21654.969,E2 21654.969} C_VEL
LIN {X 0,Y 168.984,Z 1016.575,A -85,B 0,C 180,E1 21658.413,E2 21658.413} C_VEL
LIN {X 0,Y 162.11,Z 1018.25,A -85,B 0,C 180,E1 21663.946,E2 21663.946} C_VEL
LIN {X 0,Y 156.534,Z 1018.241,A -85,B 0,C 180,E1 21669.698,E2 21669.698} C_VEL
LIN {X 0,Y 156.492,Z 1018.02,A -85,B 0,C 180,E1 21669.898,E2 21669.898} C_VEL
LIN {X 0,Y 156.491,Z 1014.528,A -85,B 0,C 180,E1 21678.841,E2 21678.841} C_VEL
LIN {X 0,Y 160.652,Z 1004.813,A -85,B 0,C 180,E1 21689.998,E2 21689.998} C_VEL
LIN {X 0,Y 168.021,Z 989.916,A -85,B 0,C 180,E1 21699.726,E2 21699.726} C_VEL
LIN {X 0,Y 177.279,Z 970.932,A -85,B 0,C 180,E1 21707.391,E2 21707.391} C_VEL
LIN {X 0,Y 184.067,Z 955.327,A -85,B 0,C 180,E1 21711.723,E2 21711.723} C_VEL
LIN {X 0,Y 183.849,Z 936.008,A -85,B 0,C 180,E1 21717.807,E2 21717.807} C_VEL
LIN {X 0,Y 182.336,Z 931.238,A -85,B 0,C 180,E1 21719.62,E2 21719.62} C_VEL
LIN {X 0,Y 169.94,Z 933.345,A -85,B 0,C 180,E1 21724.027,E2 21724.027} C_VEL
LIN {X 0,Y 170.121,Z 941.669,A -85,B 0,C 180,E1 21725.751,E2 21725.751} C_VEL
LIN {X 0,Y 164.32,Z 968.189,A -85,B 0,C 180,E1 21732.155,E2 21732.155} C_VEL
LIN {X 0,Y 159.438,Z 989.214,A -85,B 0,C 180,E1 21739.984,E2 21739.984} C_VEL
LIN {X 0,Y 156.325,Z 1005.821,A -85,B 0,C 180,E1 21749.5,E2 21749.5} C_VEL
LIN {X 0,Y 156.131,Z 1015.938,A -85,B 0,C 180,E1 21758.761,E2 21758.761} C_VEL
LIN {X 0,Y 159.721,Z 1021.911,A -85,B 0,C 180,E1 21769.147,E2 21769.147} C_VEL
LIN {X 0,Y 166.642,Z 1022.694,A -85,B 0,C 180,E1 21778.026,E2 21778.026} C_VEL
LIN {X 0,Y 178.579,Z 1018.096,A -85,B 0,C 180,E1 21787.366,E2 21787.366} C_VEL
LIN {X 0,Y 194.027,Z 1007.43,A -85,B 0,C 180,E1 21795.291,E2 21795.291} C_VEL
LIN {X 0,Y 209.957,Z 991.965,A -85,B 0,C 180,E1 21801.182,E2 21801.182} C_VEL
LIN {X 0,Y 224.185,Z 973.569,A -85,B 0,C 180,E1 21805.545,E2 21805.545} C_VEL
LIN {X 0,Y 226.802,Z 969.014,A -85,B 0,C 180,E1 21807.902,E2 21807.902} C_VEL
